KUKA KRL program: EPS_2_25252_SD6_A_20250910061732.src

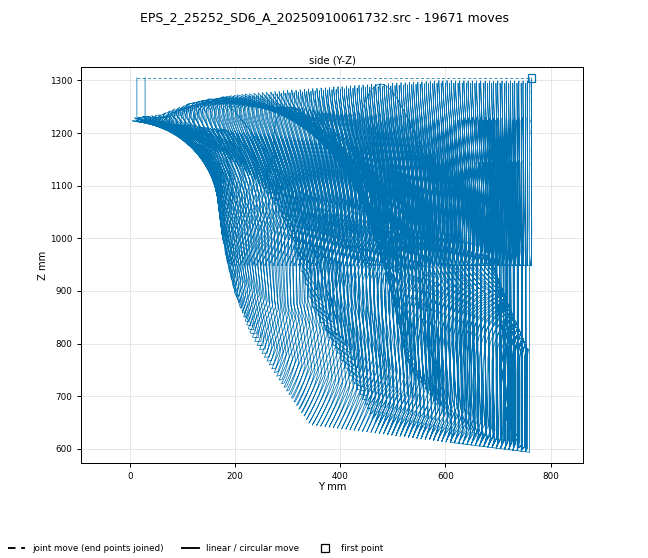
[picture p0: tool path of EPS_2_25252_SD6_A_20250910061732.src, 19671 of 19673 moves have a stored position in this frame; points joined in program order, loops and branches not executed]
&ACCESS RVP
&REL 4
&COMMENT QRS 19112012
&PARAM EDITMASK = *
DEF PART()
EXT BAS (BAS_COMMAND :IN,REAL :IN )
INT I
BAS (#INITMOV,0 )

;KUKA QRS Post kuka4.cps  Date:22-06-2017 !

File_ID=2834

QRS_PRE_INIT()

;Init var - Until changes are made in qrs_pre_init
Outlet_Square_prg=0
Inlet_1_Square_prg=0
Inlet_2_Square_prg=0
Inlet_3_Square_prg=0
Inlet_4_Square_prg=0
Inlet_5_Square_prg=0

Outlet_1={X 0.000, Y 582.000, Z 990.000, B 0.000, E1 0.000 }
Inlet_1={X 0.000, Y 651.840, Z 887.500, B 0.000, E1 181.000 }
Inlet_2={X 0.000, Y 582.000, Z 920.000, B 0.000, E1 273.000 }
Outlet_1_type=610
Inlet_1_type=299
Inlet_2_type=610
;QRS#1=Sidecore dimensions
;QRS#2=600-24" Concrete
;QRS#3=300-12" PVC SDR 35
;QRS#4=600-24" Concrete
;QRS#5=
;QRS#6=
;QRS#7=
;QRS#8=
;QRS#9=S306-34L
;QRS#10=16M PSX
;QRS#11=S306-34L
;QRS#12=
;QRS#13=
;QRS#14=
;QRS#15=
;QRS#16=1524x152x1753 5,75'
;QRS#17=EPS Height
;QRS#18=1295
;QRS#19=*
;QRS#20= UPDATED VERSION 22-06-2017
;QRS#21=*
Outlet_Square=0450
Inlet_1_Square=0150
Inlet_2_Square=0450
Inlet_3_Square=0
Inlet_4_Square=0
Inlet_5_Square=0
Mill_Square=1
Outlet_Square_Prg=264
Inlet_1_Square_prg=206
Inlet_2_Square_prg=264

QRS_INIT()

$ADVANCE=5

; T1
PTP {E1 176.595,E2 176.595}
PTP {X 0,Y 763.416,A -85,B 0,C 180,E1 176.595,E2 176.595,E3 0,E4 0,E5 0,E6 0}
QRS_SPEED_INIT()
LIN {X 0,Y 763.416,Z 1305,A -85,B 0,C 180,E1 176.595,E2 176.595,E3 0,E4 0,E5 0,E6 0} C_VEL
LIN {X 0,Y 763.416,Z 950.94,A -85,B 0,C 180,E1 176.595,E2 176.595} C_VEL
LIN {X 0,Y 763.526,Z 948.94,A -85,B 0,C 180,E1 176.744,E2 176.744} C_VEL
LIN {X 0,Y 763.879,Z 948.94,A -85,B 0,C 180,E1 177.187,E2 177.187} C_VEL
LIN {X 0,Y 763.856,Z 948.94,A -85,B 0,C 180,E1 184.692,E2 184.692} C_VEL
LIN {X 0,Y 763.844,Z 948.94,A -85,B 0,C 180,E1 192.28,E2 192.28} C_VEL
LIN {X 0,Y 763.822,Z 948.94,A -85,B 0,C 180,E1 200.096,E2 200.096} C_VEL
LIN {X 0,Y 763.802,Z 948.94,A -85,B 0,C 180,E1 208.326,E2 208.326} C_VEL
LIN {X 0,Y 762.908,Z 948.94,A -85,B 0,C 180,E1 213.344,E2 213.344} C_VEL
LIN {X 0,Y 763.801,Z 948.94,A -85,B 0,C 180,E1 214.936,E2 214.936} C_VEL
LIN {X 0,Y 762.569,Z 948.94,A -85,B 0,C 180,E1 217.327,E2 217.327} C_VEL
LIN {X 0,Y 763.787,Z 948.94,A -85,B 0,C 180,E1 222.132,E2 222.132} C_VEL
LIN {X 0,Y 763.6,Z 948.94,A -85,B 0,C 180,E1 222.571,E2 222.571} C_VEL
LIN {X 0,Y 763.857,Z 948.94,A -85,B 0,C 180,E1 230.259,E2 230.259} C_VEL
LIN {X 0,Y 763.749,Z 948.94,A -85,B 0,C 180,E1 236.564,E2 236.564} C_VEL
LIN {X 0,Y 763.497,Z 948.94,A -85,B 0,C 180,E1 237.308,E2 237.308} C_VEL
LIN {X 0,Y 763.827,Z 948.94,A -85,B 0,C 180,E1 243.397,E2 243.397} C_VEL
LIN {X 0,Y 763.404,Z 948.94,A -85,B 0,C 180,E1 243.594,E2 243.594} C_VEL
LIN {X 0,Y 763.701,Z 1010.798,A -85,B 0,C 180,E1 244.25,E2 244.25} C_VEL
LIN {X 0,Y 763.661,Z 1023.487,A -85,B 0,C 180,E1 244.413,E2 244.413} C_VEL
LIN {X 0,Y 763.555,Z 1034.565,A -85,B 0,C 180,E1 244.586,E2 244.586} C_VEL
LIN {X 0,Y 763.798,Z 1053.031,A -85,B 0,C 180,E1 244.967,E2 244.967} C_VEL
LIN {X 0,Y 763.799,Z 1068.002,A -85,B 0,C 180,E1 245.336,E2 245.336} C_VEL
LIN {X 0,Y 763.786,Z 1082.074,A -85,B 0,C 180,E1 245.738,E2 245.738} C_VEL
LIN {X 0,Y 763.598,Z 1095.558,A -85,B 0,C 180,E1 246.171,E2 246.171} C_VEL
LIN {X 0,Y 763.732,Z 1110.988,A -85,B 0,C 180,E1 246.751,E2 246.751} C_VEL
LIN {X 0,Y 763.705,Z 1123.304,A -85,B 0,C 180,E1 247.259,E2 247.259} C_VEL
LIN {X 0,Y 763.746,Z 1137.059,A -85,B 0,C 180,E1 247.894,E2 247.894} C_VEL
LIN {X 0,Y 763.694,Z 1150.472,A -85,B 0,C 180,E1 248.578,E2 248.578} C_VEL
LIN {X 0,Y 763.632,Z 1163.214,A -85,B 0,C 180,E1 249.293,E2 249.293} C_VEL
LIN {X 0,Y 763.454,Z 1174.901,A -85,B 0,C 180,E1 250.006,E2 250.006} C_VEL
LIN {X 0,Y 763.487,Z 1186.338,A -85,B 0,C 180,E1 250.774,E2 250.774} C_VEL
LIN {X 0,Y 763.678,Z 1195.926,A -85,B 0,C 180,E1 251.472,E2 251.472} C_VEL
LIN {X 0,Y 763.773,Z 1205.944,A -85,B 0,C 180,E1 252.258,E2 252.258} C_VEL
LIN {X 0,Y 763.425,Z 1217.367,A -85,B 0,C 180,E1 253.232,E2 253.232} C_VEL
LIN {X 0,Y 763.24,Z 1226.789,A -85,B 0,C 180,E1 254.111,E2 254.111} C_VEL
LIN {X 0,Y 763.374,Z 1235.4,A -85,B 0,C 180,E1 254.99,E2 254.99} C_VEL
LIN {X 0,Y 763.744,Z 1243.954,A -85,B 0,C 180,E1 255.948,E2 255.948} C_VEL
LIN {X 0,Y 763.788,Z 1247.786,A -85,B 0,C 180,E1 256.411,E2 256.411} C_VEL
LIN {X 0,Y 763.506,Z 1252.144,A -85,B 0,C 180,E1 256.944,E2 256.944} C_VEL
LIN {X 0,Y 763.029,Z 1259.656,A -85,B 0,C 180,E1 257.948,E2 257.948} C_VEL
LIN {X 0,Y 762.924,Z 1266.105,A -85,B 0,C 180,E1 258.904,E2 258.904} C_VEL
LIN {X 0,Y 763.387,Z 1273.197,A -85,B 0,C 180,E1 260.104,E2 260.104} C_VEL
LIN {X 0,Y 763.861,Z 1278.258,A -85,B 0,C 180,E1 261.06,E2 261.06} C_VEL
LIN {X 0,Y 763.274,Z 1282.688,A -85,B 0,C 180,E1 262.001,E2 262.001} C_VEL
LIN {X 0,Y 762.799,Z 1286.562,A -85,B 0,C 180,E1 262.943,E2 262.943} C_VEL
LIN {X 0,Y 762.692,Z 1288.341,A -85,B 0,C 180,E1 263.415,E2 263.415} C_VEL
LIN {X 0,Y 762.777,Z 1291.504,A -85,B 0,C 180,E1 264.36,E2 264.36} C_VEL
LIN {X 0,Y 763.282,Z 1294.069,A -85,B 0,C 180,E1 265.305,E2 265.305} C_VEL
LIN {X 0,Y 763.855,Z 1296.057,A -85,B 0,C 180,E1 266.211,E2 266.211} C_VEL
LIN {X 0,Y 763.535,Z 1297.167,A -85,B 0,C 180,E1 266.77,E2 266.77} C_VEL
LIN {X 0,Y 762.865,Z 1298.824,A -85,B 0,C 180,E1 267.936,E2 267.936} C_VEL
LIN {X 0,Y 762.698,Z 1299.723,A -85,B 0,C 180,E1 269.062,E2 269.062} C_VEL
LIN {X 0,Y 763.57,Z 1299.689,A -85,B 0,C 180,E1 270.939,E2 270.939} C_VEL
LIN {X 0,Y 763.743,Z 1299.172,A -85,B 0,C 180,E1 271.626,E2 271.626} C_VEL
LIN {X 0,Y 763.022,Z 1297.802,A -85,B 0,C 180,E1 272.817,E2 272.817} C_VEL
LIN {X 0,Y 762.7,Z 1296.172,A -85,B 0,C 180,E1 273.759,E2 273.759} C_VEL
LIN {X 0,Y 762.79,Z 1294.072,A -85,B 0,C 180,E1 274.7,E2 274.7} C_VEL
LIN {X 0,Y 763.256,Z 1291.49,A -85,B 0,C 180,E1 275.639,E2 275.639} C_VEL
LIN {X 0,Y 763.854,Z 1288.314,A -85,B 0,C 180,E1 276.577,E2 276.577} C_VEL
LIN {X 0,Y 763.331,Z 1284.657,A -85,B 0,C 180,E1 277.527,E2 277.527} C_VEL
LIN {X 0,Y 762.963,Z 1281.571,A -85,B 0,C 180,E1 278.241,E2 278.241} C_VEL
LIN {X 0,Y 762.777,Z 1278.249,A -85,B 0,C 180,E1 278.955,E2 278.955} C_VEL
LIN {X 0,Y 763.033,Z 1271.861,A -85,B 0,C 180,E1 280.142,E2 280.142} C_VEL
LIN {X 0,Y 763.586,Z 1266.091,A -85,B 0,C 180,E1 281.088,E2 281.088} C_VEL
LIN {X 0,Y 763.837,Z 1262.881,A -85,B 0,C 180,E1 281.563,E2 281.563} C_VEL
LIN {X 0,Y 763.471,Z 1257.055,A -85,B 0,C 180,E1 282.404,E2 282.404} C_VEL
LIN {X 0,Y 763.075,Z 1250.184,A -85,B 0,C 180,E1 283.313,E2 283.313} C_VEL
LIN {X 0,Y 763.016,Z 1242.631,A -85,B 0,C 180,E1 284.223,E2 284.223} C_VEL
LIN {X 0,Y 763.396,Z 1233.611,A -85,B 0,C 180,E1 285.201,E2 285.201} C_VEL
LIN {X 0,Y 763.805,Z 1223.978,A -85,B 0,C 180,E1 286.151,E2 286.151} C_VEL
LIN {X 0,Y 763.566,Z 1214.615,A -85,B 0,C 180,E1 287.012,E2 287.012} C_VEL
LIN {X 0,Y 763.309,Z 1204.368,A -85,B 0,C 180,E1 287.878,E2 287.878} C_VEL
LIN {X 0,Y 763.361,Z 1193.883,A -85,B 0,C 180,E1 288.687,E2 288.687} C_VEL
LIN {X 0,Y 763.618,Z 1182.933,A -85,B 0,C 180,E1 289.459,E2 289.459} C_VEL
LIN {X 0,Y 763.758,Z 1171.052,A -85,B 0,C 180,E1 290.229,E2 290.229} C_VEL
LIN {X 0,Y 763.669,Z 1158.921,A -85,B 0,C 180,E1 290.955,E2 290.955} C_VEL
LIN {X 0,Y 763.569,Z 1146.964,A -85,B 0,C 180,E1 291.612,E2 291.612} C_VEL
LIN {X 0,Y 763.634,Z 1134.379,A -85,B 0,C 180,E1 292.238,E2 292.238} C_VEL
LIN {X 0,Y 763.716,Z 1120.252,A -85,B 0,C 180,E1 292.87,E2 292.87} C_VEL
LIN {X 0,Y 763.734,Z 1110.933,A -85,B 0,C 180,E1 293.252,E2 293.252} C_VEL
LIN {X 0,Y 763.776,Z 1095.487,A -85,B 0,C 180,E1 293.826,E2 293.826} C_VEL
LIN {X 0,Y 763.739,Z 1080.093,A -85,B 0,C 180,E1 294.326,E2 294.326} C_VEL
LIN {X 0,Y 763.763,Z 1063.413,A -85,B 0,C 180,E1 294.785,E2 294.785} C_VEL
LIN {X 0,Y 763.546,Z 1049.599,A -85,B 0,C 180,E1 295.119,E2 295.119} C_VEL
LIN {X 0,Y 763.829,Z 1033.797,A -85,B 0,C 180,E1 295.417,E2 295.417} C_VEL
LIN {X 0,Y 763.825,Z 1018.657,A -85,B 0,C 180,E1 295.65,E2 295.65} C_VEL
LIN {X 0,Y 763.807,Z 1000.838,A -85,B 0,C 180,E1 295.857,E2 295.857} C_VEL
LIN {X 0,Y 763.398,Z 948.94,A -85,B 0,C 180,E1 296.405,E2 296.405} C_VEL
LIN {X 0,Y 763.703,Z 948.94,A -85,B 0,C 180,E1 296.465,E2 296.465} C_VEL
LIN {X 0,Y 763.627,Z 948.94,A -85,B 0,C 180,E1 297.495,E2 297.495} C_VEL
LIN {X 0,Y 763.6,Z 948.94,A -85,B 0,C 180,E1 298.335,E2 298.335} C_VEL
LIN {X 0,Y 763.684,Z 948.94,A -85,B 0,C 180,E1 299.853,E2 299.853} C_VEL
LIN {X 0,Y 763.798,Z 948.94,A -85,B 0,C 180,E1 307.257,E2 307.257} C_VEL
LIN {X 0,Y 762.303,Z 948.94,A -85,B 0,C 180,E1 312.462,E2 312.462} C_VEL
LIN {X 0,Y 763.54,Z 948.94,A -85,B 0,C 180,E1 314.733,E2 314.733} C_VEL
LIN {X 0,Y 763.758,Z 948.94,A -85,B 0,C 180,E1 315.284,E2 315.284} C_VEL
LIN {X 0,Y 763.727,Z 948.94,A -85,B 0,C 180,E1 323.303,E2 323.303} C_VEL
LIN {X 0,Y 762.819,Z 948.94,A -85,B 0,C 180,E1 325.013,E2 325.013} C_VEL
LIN {X 0,Y 763.876,Z 948.94,A -85,B 0,C 180,E1 330.979,E2 330.979} C_VEL
LIN {X 0,Y 762.688,Z 948.94,A -85,B 0,C 180,E1 331.215,E2 331.215} C_VEL
LIN {X 0,Y 762.37,Z 948.94,A -85,B 0,C 180,E1 331.237,E2 331.237} C_VEL
LIN {X 0,Y 762.335,Z 950.241,A -85,B 0,C 180,E1 331.271,E2 331.271} C_VEL
LIN {X 0,Y 763.361,Z 966.778,A -85,B 0,C 180,E1 331.573,E2 331.573} C_VEL
LIN {X 0,Y 763.732,Z 983.068,A -85,B 0,C 180,E1 331.92,E2 331.92} C_VEL
LIN {X 0,Y 763.791,Z 997.305,A -85,B 0,C 180,E1 332.271,E2 332.271} C_VEL
LIN {X 0,Y 763.798,Z 1012.281,A -85,B 0,C 180,E1 332.701,E2 332.701} C_VEL
LIN {X 0,Y 763.667,Z 1027.209,A -85,B 0,C 180,E1 333.189,E2 333.189} C_VEL
LIN {X 0,Y 763.708,Z 1041.233,A -85,B 0,C 180,E1 333.715,E2 333.715} C_VEL
LIN {X 0,Y 763.614,Z 1054.77,A -85,B 0,C 180,E1 334.278,E2 334.278} C_VEL
LIN {X 0,Y 763.605,Z 1067.742,A -85,B 0,C 180,E1 334.879,E2 334.879} C_VEL
LIN {X 0,Y 763.72,Z 1080.324,A -85,B 0,C 180,E1 335.525,E2 335.525} C_VEL
LIN {X 0,Y 763.702,Z 1092.995,A -85,B 0,C 180,E1 336.237,E2 336.237} C_VEL
LIN {X 0,Y 763.572,Z 1103.494,A -85,B 0,C 180,E1 336.871,E2 336.871} C_VEL
LIN {X 0,Y 763.366,Z 1114.975,A -85,B 0,C 180,E1 337.628,E2 337.628} C_VEL
LIN {X 0,Y 763.422,Z 1126.864,A -85,B 0,C 180,E1 338.494,E2 338.494} C_VEL
LIN {X 0,Y 763.687,Z 1137.376,A -85,B 0,C 180,E1 339.333,E2 339.333} C_VEL
LIN {X 0,Y 763.755,Z 1146.543,A -85,B 0,C 180,E1 340.119,E2 340.119} C_VEL
LIN {X 0,Y 763.366,Z 1156.466,A -85,B 0,C 180,E1 341.036,E2 341.036} C_VEL
LIN {X 0,Y 763.138,Z 1164.781,A -85,B 0,C 180,E1 341.872,E2 341.872} C_VEL
LIN {X 0,Y 763.296,Z 1173.673,A -85,B 0,C 180,E1 342.86,E2 342.86} C_VEL
LIN {X 0,Y 763.713,Z 1181.74,A -85,B 0,C 180,E1 343.848,E2 343.848} C_VEL
LIN {X 0,Y 763.782,Z 1185.725,A -85,B 0,C 180,E1 344.38,E2 344.38} C_VEL
LIN {X 0,Y 763.393,Z 1190.811,A -85,B 0,C 180,E1 345.08,E2 345.08} C_VEL
LIN {X 0,Y 763.022,Z 1195.576,A -85,B 0,C 180,E1 345.778,E2 345.778} C_VEL
LIN {X 0,Y 762.856,Z 1202.68,A -85,B 0,C 180,E1 346.955,E2 346.955} C_VEL
LIN {X 0,Y 763.206,Z 1207.972,A -85,B 0,C 180,E1 347.949,E2 347.949} C_VEL
LIN {X 0,Y 763.862,Z 1213.536,A -85,B 0,C 180,E1 349.155,E2 349.155} C_VEL
LIN {X 0,Y 763.274,Z 1217.354,A -85,B 0,C 180,E1 350.101,E2 350.101} C_VEL
LIN {X 0,Y 762.801,Z 1220.606,A -85,B 0,C 180,E1 351.046,E2 351.046} C_VEL
LIN {X 0,Y 762.674,Z 1222.073,A -85,B 0,C 180,E1 351.519,E2 351.519} C_VEL
LIN {X 0,Y 762.784,Z 1224.641,A -85,B 0,C 180,E1 352.469,E2 352.469} C_VEL
LIN {X 0,Y 763.298,Z 1226.62,A -85,B 0,C 180,E1 353.419,E2 353.419} C_VEL
LIN {X 0,Y 763.877,Z 1228.101,A -85,B 0,C 180,E1 354.367,E2 354.367} C_VEL
LIN {X 0,Y 763.297,Z 1229.174,A -85,B 0,C 180,E1 355.304,E2 355.304} C_VEL
LIN {X 0,Y 762.81,Z 1229.786,A -85,B 0,C 180,E1 356.243,E2 356.243} C_VEL
LIN {X 0,Y 762.699,Z 1229.932,A -85,B 0,C 180,E1 357.182,E2 357.182} C_VEL
LIN {X 0,Y 762.878,Z 1229.741,A -85,B 0,C 180,E1 357.815,E2 357.815} C_VEL
LIN {X 0,Y 763.571,Z 1228.757,A -85,B 0,C 180,E1 359.062,E2 359.062} C_VEL
LIN {X 0,Y 763.711,Z 1227.71,A -85,B 0,C 180,E1 359.812,E2 359.812} C_VEL
LIN {X 0,Y 763.226,Z 1226.472,A -85,B 0,C 180,E1 360.563,E2 360.563} C_VEL
LIN {X 0,Y 762.773,Z 1224.607,A -85,B 0,C 180,E1 361.456,E2 361.456} C_VEL
LIN {X 0,Y 762.819,Z 1220.763,A -85,B 0,C 180,E1 362.817,E2 362.817} C_VEL
LIN {X 0,Y 763.286,Z 1217.571,A -85,B 0,C 180,E1 363.755,E2 363.755} C_VEL
LIN {X 0,Y 763.871,Z 1213.785,A -85,B 0,C 180,E1 364.692,E2 364.692} C_VEL
LIN {X 0,Y 763.266,Z 1208.395,A -85,B 0,C 180,E1 365.873,E2 365.873} C_VEL
LIN {X 0,Y 762.935,Z 1202.109,A -85,B 0,C 180,E1 367.057,E2 367.057} C_VEL
LIN {X 0,Y 763.249,Z 1194.841,A -85,B 0,C 180,E1 368.237,E2 368.237} C_VEL
LIN {X 0,Y 763.726,Z 1188.367,A -85,B 0,C 180,E1 369.18,E2 369.18} C_VEL
LIN {X 0,Y 763.833,Z 1186.575,A -85,B 0,C 180,E1 369.416,E2 369.416} C_VEL
LIN {X 0,Y 763.53,Z 1181.216,A -85,B 0,C 180,E1 370.134,E2 370.134} C_VEL
LIN {X 0,Y 763.074,Z 1172.289,A -85,B 0,C 180,E1 371.214,E2 371.214} C_VEL
LIN {X 0,Y 763.072,Z 1163.507,A -85,B 0,C 180,E1 372.173,E2 372.173} C_VEL
LIN {X 0,Y 763.482,Z 1153.382,A -85,B 0,C 180,E1 373.167,E2 373.167} C_VEL
LIN {X 0,Y 763.794,Z 1145.374,A -85,B 0,C 180,E1 373.897,E2 373.897} C_VEL
LIN {X 0,Y 763.543,Z 1133.799,A -85,B 0,C 180,E1 374.872,E2 374.872} C_VEL
LIN {X 0,Y 763.312,Z 1124.099,A -85,B 0,C 180,E1 375.628,E2 375.628} C_VEL
LIN {X 0,Y 763.349,Z 1113.189,A -85,B 0,C 180,E1 376.404,E2 376.404} C_VEL
LIN {X 0,Y 763.612,Z 1100.958,A -85,B 0,C 180,E1 377.194,E2 377.194} C_VEL
LIN {X 0,Y 763.732,Z 1088.56,A -85,B 0,C 180,E1 377.929,E2 377.929} C_VEL
LIN {X 0,Y 763.702,Z 1076.06,A -85,B 0,C 180,E1 378.609,E2 378.609} C_VEL
LIN {X 0,Y 763.59,Z 1064.721,A -85,B 0,C 180,E1 379.179,E2 379.179} C_VEL
LIN {X 0,Y 763.625,Z 1050.751,A -85,B 0,C 180,E1 379.808,E2 379.808} C_VEL
LIN {X 0,Y 763.711,Z 1036.783,A -85,B 0,C 180,E1 380.369,E2 380.369} C_VEL
LIN {X 0,Y 763.667,Z 1025.67,A -85,B 0,C 180,E1 380.777,E2 380.777} C_VEL
LIN {X 0,Y 763.756,Z 1008.064,A -85,B 0,C 180,E1 381.338,E2 381.338} C_VEL
LIN {X 0,Y 763.736,Z 993.52,A -85,B 0,C 180,E1 381.739,E2 381.739} C_VEL
LIN {X 0,Y 763.708,Z 978.398,A -85,B 0,C 180,E1 382.093,E2 382.093} C_VEL
LIN {X 0,Y 763.357,Z 963.499,A -85,B 0,C 180,E1 382.393,E2 382.393} C_VEL
LIN {X 0,Y 762.407,Z 950.883,A -85,B 0,C 180,E1 382.628,E2 382.628} C_VEL
LIN {X 0,Y 762.139,Z 949.021,A -85,B 0,C 180,E1 382.661,E2 382.661} C_VEL
LIN {X 0,Y 763.124,Z 948.94,A -85,B 0,C 180,E1 382.74,E2 382.74} C_VEL
LIN {X 0,Y 763.665,Z 948.94,A -85,B 0,C 180,E1 383.269,E2 383.269} C_VEL
LIN {X 0,Y 763.828,Z 948.94,A -85,B 0,C 180,E1 388.325,E2 388.325} C_VEL
LIN {X 0,Y 762.698,Z 948.94,A -85,B 0,C 180,E1 394.994,E2 394.994} C_VEL
LIN {X 0,Y 763.702,Z 948.94,A -85,B 0,C 180,E1 396.695,E2 396.695} C_VEL
LIN {X 0,Y 763.721,Z 948.94,A -85,B 0,C 180,E1 404.719,E2 404.719} C_VEL
LIN {X 0,Y 763.507,Z 948.94,A -85,B 0,C 180,E1 405.265,E2 405.265} C_VEL
LIN {X 0,Y 762.431,Z 948.94,A -85,B 0,C 180,E1 410.388,E2 410.388} C_VEL
LIN {X 0,Y 763.801,Z 948.94,A -85,B 0,C 180,E1 412.743,E2 412.743} C_VEL
LIN {X 0,Y 763.669,Z 948.94,A -85,B 0,C 180,E1 420.149,E2 420.149} C_VEL
LIN {X 0,Y 762.955,Z 948.94,A -85,B 0,C 180,E1 421.639,E2 421.639} C_VEL
LIN {X 0,Y 763.83,Z 948.94,A -85,B 0,C 180,E1 427.894,E2 427.894} C_VEL
LIN {X 0,Y 763.858,Z 948.94,A -85,B 0,C 180,E1 434.777,E2 434.777} C_VEL
LIN {X 0,Y 763.313,Z 948.94,A -85,B 0,C 180,E1 434.94,E2 434.94} C_VEL
LIN {X 0,Y 762.376,Z 948.94,A -85,B 0,C 180,E1 435.024,E2 435.024} C_VEL
LIN {X 0,Y 763.453,Z 975.866,A -85,B 0,C 180,E1 435.303,E2 435.303} C_VEL
LIN {X 0,Y 763.818,Z 998.319,A -85,B 0,C 180,E1 435.532,E2 435.532} C_VEL
LIN {X 0,Y 763.817,Z 1010.228,A -85,B 0,C 180,E1 435.708,E2 435.708} C_VEL
LIN {X 0,Y 763.804,Z 1018.714,A -85,B 0,C 180,E1 435.874,E2 435.874} C_VEL
LIN {X 0,Y 763.805,Z 1028.192,A -85,B 0,C 180,E1 436.1,E2 436.1} C_VEL
LIN {X 0,Y 763.731,Z 1036.369,A -85,B 0,C 180,E1 436.329,E2 436.329} C_VEL
LIN {X 0,Y 763.74,Z 1044.631,A -85,B 0,C 180,E1 436.598,E2 436.598} C_VEL
LIN {X 0,Y 763.845,Z 1054.622,A -85,B 0,C 180,E1 436.974,E2 436.974} C_VEL
LIN {X 0,Y 763.835,Z 1063.932,A -85,B 0,C 180,E1 437.383,E2 437.383} C_VEL
LIN {X 0,Y 763.698,Z 1071.923,A -85,B 0,C 180,E1 437.777,E2 437.777} C_VEL
LIN {X 0,Y 763.546,Z 1079.501,A -85,B 0,C 180,E1 438.194,E2 438.194} C_VEL
LIN {X 0,Y 763.575,Z 1087.281,A -85,B 0,C 180,E1 438.673,E2 438.673} C_VEL
LIN {X 0,Y 763.799,Z 1095.832,A -85,B 0,C 180,E1 439.273,E2 439.273} C_VEL
LIN {X 0,Y 763.835,Z 1101.944,A -85,B 0,C 180,E1 439.75,E2 439.75} C_VEL
LIN {X 0,Y 763.6,Z 1107.496,A -85,B 0,C 180,E1 440.223,E2 440.223} C_VEL
LIN {X 0,Y 763.321,Z 1112.557,A -85,B 0,C 180,E1 440.695,E2 440.695} C_VEL
LIN {X 0,Y 763.183,Z 1117.18,A -85,B 0,C 180,E1 441.168,E2 441.168} C_VEL
LIN {X 0,Y 763.261,Z 1121.403,A -85,B 0,C 180,E1 441.644,E2 441.644} C_VEL
LIN {X 0,Y 763.56,Z 1126.164,A -85,B 0,C 180,E1 442.239,E2 442.239} C_VEL
LIN {X 0,Y 763.801,Z 1129.593,A -85,B 0,C 180,E1 442.714,E2 442.714} C_VEL
LIN {X 0,Y 763.871,Z 1131.208,A -85,B 0,C 180,E1 442.951,E2 442.951} C_VEL
LIN {X 0,Y 763.472,Z 1135.557,A -85,B 0,C 180,E1 443.655,E2 443.655} C_VEL
LIN {X 0,Y 763.096,Z 1139.231,A -85,B 0,C 180,E1 444.36,E2 444.36} C_VEL
LIN {X 0,Y 763.009,Z 1141.39,A -85,B 0,C 180,E1 444.831,E2 444.831} C_VEL
LIN {X 0,Y 763.112,Z 1143.271,A -85,B 0,C 180,E1 445.302,E2 445.302} C_VEL
LIN {X 0,Y 763.388,Z 1145.04,A -85,B 0,C 180,E1 445.823,E2 445.823} C_VEL
LIN {X 0,Y 763.774,Z 1146.85,A -85,B 0,C 180,E1 446.466,E2 446.466} C_VEL
LIN {X 0,Y 763.607,Z 1148.403,A -85,B 0,C 180,E1 447.185,E2 447.185} C_VEL
LIN {X 0,Y 763.131,Z 1149.434,A -85,B 0,C 180,E1 447.934,E2 447.934} C_VEL
LIN {X 0,Y 762.969,Z 1149.77,A -85,B 0,C 180,E1 448.309,E2 448.309} C_VEL
LIN {X 0,Y 762.962,Z 1149.961,A -85,B 0,C 180,E1 449.06,E2 449.06} C_VEL
LIN {X 0,Y 763.329,Z 1149.57,A -85,B 0,C 180,E1 449.811,E2 449.811} C_VEL
LIN {X 0,Y 763.801,Z 1148.636,A -85,B 0,C 180,E1 450.561,E2 450.561} C_VEL
LIN {X 0,Y 763.769,Z 1147.968,A -85,B 0,C 180,E1 450.936,E2 450.936} C_VEL
LIN {X 0,Y 763.177,Z 1145.441,A -85,B 0,C 180,E1 451.97,E2 451.97} C_VEL
LIN {X 0,Y 763.031,Z 1143.772,A -85,B 0,C 180,E1 452.471,E2 452.471} C_VEL
LIN {X 0,Y 763.126,Z 1141.244,A -85,B 0,C 180,E1 453.114,E2 453.114} C_VEL
LIN {X 0,Y 763.441,Z 1138.352,A -85,B 0,C 180,E1 453.733,E2 453.733} C_VEL
LIN {X 0,Y 763.825,Z 1134.861,A -85,B 0,C 180,E1 454.371,E2 454.371} C_VEL
LIN {X 0,Y 763.669,Z 1131.439,A -85,B 0,C 180,E1 454.927,E2 454.927} C_VEL
LIN {X 0,Y 763.323,Z 1126.447,A -85,B 0,C 180,E1 455.636,E2 455.636} C_VEL
LIN {X 0,Y 763.231,Z 1120.749,A -85,B 0,C 180,E1 456.344,E2 456.344} C_VEL
LIN {X 0,Y 763.532,Z 1114.219,A -85,B 0,C 180,E1 457.05,E2 457.05} C_VEL
LIN {X 0,Y 763.832,Z 1108.014,A -85,B 0,C 180,E1 457.638,E2 457.638} C_VEL
LIN {X 0,Y 763.786,Z 1102.54,A -85,B 0,C 180,E1 458.112,E2 458.112} C_VEL
LIN {X 0,Y 763.575,Z 1096.526,A -85,B 0,C 180,E1 458.588,E2 458.588} C_VEL
LIN {X 0,Y 763.441,Z 1089.89,A -85,B 0,C 180,E1 459.064,E2 459.064} C_VEL
LIN {X 0,Y 763.556,Z 1081.564,A -85,B 0,C 180,E1 459.597,E2 459.597} C_VEL
LIN {X 0,Y 763.796,Z 1073.109,A -85,B 0,C 180,E1 460.07,E2 460.07} C_VEL
LIN {X 0,Y 763.853,Z 1066.053,A -85,B 0,C 180,E1 460.426,E2 460.426} C_VEL
LIN {X 0,Y 763.8,Z 1058.187,A -85,B 0,C 180,E1 460.784,E2 460.784} C_VEL
LIN {X 0,Y 763.629,Z 1049.304,A -85,B 0,C 180,E1 461.145,E2 461.145} C_VEL
LIN {X 0,Y 763.644,Z 1038.984,A -85,B 0,C 180,E1 461.503,E2 461.503} C_VEL
LIN {X 0,Y 763.804,Z 1029.717,A -85,B 0,C 180,E1 461.77,E2 461.77} C_VEL
LIN {X 0,Y 763.777,Z 1020.573,A -85,B 0,C 180,E1 461.995,E2 461.995} C_VEL
LIN {X 0,Y 763.848,Z 1011.303,A -85,B 0,C 180,E1 462.181,E2 462.181} C_VEL
LIN {X 0,Y 763.833,Z 1000.704,A -85,B 0,C 180,E1 462.349,E2 462.349} C_VEL
LIN {X 0,Y 763.809,Z 984.227,A -85,B 0,C 180,E1 462.521,E2 462.521} C_VEL
LIN {X 0,Y 763.331,Z 953.121,A -85,B 0,C 180,E1 462.825,E2 462.825} C_VEL
LIN {X 0,Y 763.254,Z 948.94,A -85,B 0,C 180,E1 462.872,E2 462.872} C_VEL
LIN {X 0,Y 763.703,Z 948.94,A -85,B 0,C 180,E1 462.95,E2 462.95} C_VEL
LIN {X 0,Y 763.603,Z 948.94,A -85,B 0,C 180,E1 463.37,E2 463.37} C_VEL
LIN {X 0,Y 763.824,Z 948.94,A -85,B 0,C 180,E1 470.094,E2 470.094} C_VEL
LIN {X 0,Y 763.807,Z 948.94,A -85,B 0,C 180,E1 478.324,E2 478.324} C_VEL
LIN {X 0,Y 761.983,Z 948.94,A -85,B 0,C 180,E1 482.765,E2 482.765} C_VEL
LIN {X 0,Y 762.706,Z 948.94,A -85,B 0,C 180,E1 484.991,E2 484.991} C_VEL
LIN {X 0,Y 763.719,Z 948.94,A -85,B 0,C 180,E1 486.697,E2 486.697} C_VEL
LIN {X 0,Y 763.746,Z 948.94,A -85,B 0,C 180,E1 494.714,E2 494.714} C_VEL
LIN {X 0,Y 763.531,Z 948.94,A -85,B 0,C 180,E1 495.267,E2 495.267} C_VEL
LIN {X 0,Y 762.429,Z 948.94,A -85,B 0,C 180,E1 500.385,E2 500.385} C_VEL
LIN {X 0,Y 763.793,Z 948.94,A -85,B 0,C 180,E1 502.743,E2 502.743} C_VEL
LIN {X 0,Y 763.668,Z 948.94,A -85,B 0,C 180,E1 510.145,E2 510.145} C_VEL
LIN {X 0,Y 762.96,Z 948.94,A -85,B 0,C 180,E1 511.64,E2 511.64} C_VEL
LIN {X 0,Y 763.826,Z 948.94,A -85,B 0,C 180,E1 517.895,E2 517.895} C_VEL
LIN {X 0,Y 763.489,Z 948.94,A -85,B 0,C 180,E1 524.95,E2 524.95} C_VEL
LIN {X 0,Y 763.685,Z 948.94,A -85,B 0,C 180,E1 525.791,E2 525.791} C_VEL
LIN {X 0,Y 763.849,Z 948.94,A -85,B 0,C 180,E1 529.632,E2 529.632} C_VEL
LIN {X 0,Y 763.526,Z 948.94,A -85,B 0,C 180,E1 536.744,E2 536.744} C_VEL
LIN {X 0,Y 754.559,Z 948.94,A -85,B 0,C 180,E1 539.344,E2 539.344} C_VEL
LIN {X 0,Y 754.729,Z 948.94,A -85,B 0,C 180,E1 546.339,E2 546.339} C_VEL
LIN {X 0,Y 754.988,Z 948.94,A -85,B 0,C 180,E1 553.356,E2 553.356} C_VEL
LIN {X 0,Y 755.078,Z 948.94,A -85,B 0,C 180,E1 560.952,E2 560.952} C_VEL
LIN {X 0,Y 755.072,Z 948.94,A -85,B 0,C 180,E1 569.491,E2 569.491} C_VEL
LIN {X 0,Y 754.903,Z 948.94,A -85,B 0,C 180,E1 576.365,E2 576.365} C_VEL
LIN {X 0,Y 755.336,Z 948.94,A -85,B 0,C 180,E1 582.888,E2 582.888} C_VEL
LIN {X 0,Y 755.509,Z 948.94,A -85,B 0,C 180,E1 590.794,E2 590.794} C_VEL
LIN {X 0,Y 755.189,Z 948.94,A -85,B 0,C 180,E1 597.865,E2 597.865} C_VEL
LIN {X 0,Y 755.986,Z 950.766,A -85,B 0,C 180,E1 603.335,E2 603.335} C_VEL
LIN {X 0,Y 756.522,Z 1050.329,A -85,B 0,C 180,E1 604.647,E2 604.647} C_VEL
LIN {X 0,Y 756.258,Z 1115.341,A -85,B 0,C 180,E1 606.688,E2 606.688} C_VEL
LIN {X 0,Y 755.771,Z 1175.676,A -85,B 0,C 180,E1 609.845,E2 609.845} C_VEL
LIN {X 0,Y 755.412,Z 1225.871,A -85,B 0,C 180,E1 613.848,E2 613.848} C_VEL
LIN {X 0,Y 755.043,Z 1261.823,A -85,B 0,C 180,E1 618.142,E2 618.142} C_VEL
LIN {X 0,Y 755.002,Z 1285.187,A -85,B 0,C 180,E1 622.523,E2 622.523} C_VEL
LIN {X 0,Y 755.286,Z 1297.813,A -85,B 0,C 180,E1 627.15,E2 627.15} C_VEL
LIN {X 0,Y 755.662,Z 1299.126,A -85,B 0,C 180,E1 631.754,E2 631.754} C_VEL
LIN {X 0,Y 755.652,Z 1287.259,A -85,B 0,C 180,E1 636.948,E2 636.948} C_VEL
LIN {X 0,Y 755.604,Z 1259.469,A -85,B 0,C 180,E1 642.201,E2 642.201} C_VEL
LIN {X 0,Y 755.774,Z 1218.868,A -85,B 0,C 180,E1 646.803,E2 646.803} C_VEL
LIN {X 0,Y 756.05,Z 1166.963,A -85,B 0,C 180,E1 650.695,E2 650.695} C_VEL
LIN {X 0,Y 756.349,Z 1106.488,A -85,B 0,C 180,E1 653.668,E2 653.668} C_VEL
LIN {X 0,Y 756.515,Z 1039.409,A -85,B 0,C 180,E1 655.575,E2 655.575} C_VEL
LIN {X 0,Y 755.673,Z 948.94,A -85,B 0,C 180,E1 656.755,E2 656.755} C_VEL
LIN {X 0,Y 754.178,Z 948.94,A -85,B 0,C 180,E1 663.624,E2 663.624} C_VEL
LIN {X 0,Y 754.493,Z 948.94,A -85,B 0,C 180,E1 669.258,E2 669.258} C_VEL
LIN {X 0,Y 755.064,Z 948.94,A -85,B 0,C 180,E1 676.107,E2 676.107} C_VEL
LIN {X 0,Y 755.02,Z 948.94,A -85,B 0,C 180,E1 684.525,E2 684.525} C_VEL
LIN {X 0,Y 755.078,Z 949.483,A -85,B 0,C 180,E1 690.997,E2 690.997} C_VEL
LIN {X 0,Y 756.378,Z 1018.428,A -85,B 0,C 180,E1 692.648,E2 692.648} C_VEL
LIN {X 0,Y 756.117,Z 1080.659,A -85,B 0,C 180,E1 695.318,E2 695.318} C_VEL
LIN {X 0,Y 755.833,Z 1136.369,A -85,B 0,C 180,E1 699.058,E2 699.058} C_VEL
LIN {X 0,Y 755.639,Z 1180.363,A -85,B 0,C 180,E1 703.529,E2 703.529} C_VEL
LIN {X 0,Y 755.444,Z 1210.603,A -85,B 0,C 180,E1 708.421,E2 708.421} C_VEL
LIN {X 0,Y 755.447,Z 1227.166,A -85,B 0,C 180,E1 713.667,E2 713.667} C_VEL
LIN {X 0,Y 755.103,Z 1229.503,A -85,B 0,C 180,E1 718.283,E2 718.283} C_VEL
LIN {X 0,Y 755.128,Z 1218.8,A -85,B 0,C 180,E1 723.468,E2 723.468} C_VEL
LIN {X 0,Y 755.357,Z 1194.629,A -85,B 0,C 180,E1 728.388,E2 728.388} C_VEL
LIN {X 0,Y 755.603,Z 1155.266,A -85,B 0,C 180,E1 733.164,E2 733.164} C_VEL
LIN {X 0,Y 755.884,Z 1104.369,A -85,B 0,C 180,E1 737.193,E2 737.193} C_VEL
LIN {X 0,Y 756.207,Z 1043.498,A -85,B 0,C 180,E1 740.346,E2 740.346} C_VEL
LIN {X 0,Y 756.427,Z 978.742,A -85,B 0,C 180,E1 742.345,E2 742.345} C_VEL
LIN {X 0,Y 755.452,Z 948.94,A -85,B 0,C 180,E1 743.078,E2 743.078} C_VEL
LIN {X 0,Y 754.85,Z 948.94,A -85,B 0,C 180,E1 749.527,E2 749.527} C_VEL
LIN {X 0,Y 754.795,Z 948.94,A -85,B 0,C 180,E1 757.844,E2 757.844} C_VEL
LIN {X 0,Y 754.95,Z 948.94,A -85,B 0,C 180,E1 766.063,E2 766.063} C_VEL
LIN {X 0,Y 755.132,Z 948.94,A -85,B 0,C 180,E1 773.613,E2 773.613} C_VEL
LIN {X 0,Y 754.882,Z 948.94,A -85,B 0,C 180,E1 781.782,E2 781.782} C_VEL
LIN {X 0,Y 754.922,Z 948.94,A -85,B 0,C 180,E1 789.377,E2 789.377} C_VEL
LIN {X 0,Y 754.639,Z 950.118,A -85,B 0,C 180,E1 794.893,E2 794.893} C_VEL
LIN {X 0,Y 756.032,Z 1025.236,A -85,B 0,C 180,E1 795.887,E2 795.887} C_VEL
LIN {X 0,Y 755.828,Z 1071.872,A -85,B 0,C 180,E1 797.656,E2 797.656} C_VEL
LIN {X 0,Y 755.483,Z 1110.797,A -85,B 0,C 180,E1 800.434,E2 800.434} C_VEL
LIN {X 0,Y 755.339,Z 1137.046,A -85,B 0,C 180,E1 803.878,E2 803.878} C_VEL
LIN {X 0,Y 755.646,Z 1148.306,A -85,B 0,C 180,E1 807.094,E2 807.094} C_VEL
LIN {X 0,Y 755.664,Z 1147.673,A -85,B 0,C 180,E1 811.122,E2 811.122} C_VEL
LIN {X 0,Y 755.709,Z 1132.236,A -85,B 0,C 180,E1 814.866,E2 814.866} C_VEL
LIN {X 0,Y 755.816,Z 1102.715,A -85,B 0,C 180,E1 818.195,E2 818.195} C_VEL
LIN {X 0,Y 755.985,Z 1061.969,A -85,B 0,C 180,E1 820.743,E2 820.743} C_VEL
LIN {X 0,Y 756.05,Z 1014.246,A -85,B 0,C 180,E1 822.265,E2 822.265} C_VEL
LIN {X 0,Y 755.681,Z 948.94,A -85,B 0,C 180,E1 823.082,E2 823.082} C_VEL
LIN {X 0,Y 755.185,Z 948.94,A -85,B 0,C 180,E1 830.808,E2 830.808} C_VEL
LIN {X 0,Y 754.898,Z 948.94,A -85,B 0,C 180,E1 839.467,E2 839.467} C_VEL
LIN {X 0,Y 754.847,Z 948.94,A -85,B 0,C 180,E1 847.775,E2 847.775} C_VEL
LIN {X 0,Y 754.955,Z 948.94,A -85,B 0,C 180,E1 856.068,E2 856.068} C_VEL
LIN {X 0,Y 755.119,Z 948.94,A -85,B 0,C 180,E1 863.619,E2 863.619} C_VEL
LIN {X 0,Y 754.889,Z 948.94,A -85,B 0,C 180,E1 871.791,E2 871.791} C_VEL
LIN {X 0,Y 754.785,Z 948.94,A -85,B 0,C 180,E1 879.384,E2 879.384} C_VEL
LIN {X 0,Y 755.395,Z 948.94,A -85,B 0,C 180,E1 886.821,E2 886.821} C_VEL
LIN {X 0,Y 754.227,Z 948.94,A -85,B 0,C 180,E1 893.634,E2 893.634} C_VEL
LIN {X 0,Y 755.089,Z 948.94,A -85,B 0,C 180,E1 898.261,E2 898.261} C_VEL
LIN {X 0,Y 754.559,Z 948.94,A -85,B 0,C 180,E1 899.344,E2 899.344} C_VEL
LIN {X 0,Y 746.381,Z 948.94,A -85,B 0,C 180,E1 901.974,E2 901.974} C_VEL
LIN {X 0,Y 746.272,Z 948.94,A -85,B 0,C 180,E1 907.585,E2 907.585} C_VEL
LIN {X 0,Y 746.888,Z 948.94,A -85,B 0,C 180,E1 913.503,E2 913.503} C_VEL
LIN {X 0,Y 747.18,Z 948.94,A -85,B 0,C 180,E1 920.811,E2 920.811} C_VEL
LIN {X 0,Y 747.51,Z 948.94,A -85,B 0,C 180,E1 928.487,E2 928.487} C_VEL
LIN {X 0,Y 747.468,Z 948.94,A -85,B 0,C 180,E1 935.347,E2 935.347} C_VEL
LIN {X 0,Y 747.347,Z 948.94,A -85,B 0,C 180,E1 942.856,E2 942.856} C_VEL
LIN {X 0,Y 747.013,Z 948.94,A -85,B 0,C 180,E1 951.758,E2 951.758} C_VEL
LIN {X 0,Y 746.804,Z 948.94,A -85,B 0,C 180,E1 958.83,E2 958.83} C_VEL
LIN {X 0,Y 747.641,Z 949.984,A -85,B 0,C 180,E1 963.005,E2 963.005} C_VEL
LIN {X 0,Y 749.261,Z 1051.983,A -85,B 0,C 180,E1 964.421,E2 964.421} C_VEL
LIN {X 0,Y 748.787,Z 1117.47,A -85,B 0,C 180,E1 966.53,E2 966.53} C_VEL
LIN {X 0,Y 748.074,Z 1176.827,A -85,B 0,C 180,E1 969.706,E2 969.706} C_VEL
LIN {X 0,Y 747.578,Z 1225.875,A -85,B 0,C 180,E1 973.674,E2 973.674} C_VEL
LIN {X 0,Y 747.109,Z 1261.826,A -85,B 0,C 180,E1 978.015,E2 978.015} C_VEL
LIN {X 0,Y 747.042,Z 1285.188,A -85,B 0,C 180,E1 982.443,E2 982.443} C_VEL
LIN {X 0,Y 747.327,Z 1297.816,A -85,B 0,C 180,E1 987.119,E2 987.119} C_VEL
LIN {X 0,Y 747.638,Z 1299.129,A -85,B 0,C 180,E1 991.773,E2 991.773} C_VEL
LIN {X 0,Y 747.608,Z 1287.258,A -85,B 0,C 180,E1 997.023,E2 997.023} C_VEL
LIN {X 0,Y 747.63,Z 1259.472,A -85,B 0,C 180,E1 1002.333,E2 1002.333} C_VEL
LIN {X 0,Y 747.931,Z 1218.873,A -85,B 0,C 180,E1 1006.985,E2 1006.985} C_VEL
LIN {X 0,Y 748.38,Z 1167.417,A -85,B 0,C 180,E1 1010.89,E2 1010.89} C_VEL
LIN {X 0,Y 748.918,Z 1106.901,A -85,B 0,C 180,E1 1013.901,E2 1013.901} C_VEL
LIN {X 0,Y 749.283,Z 1040.606,A -85,B 0,C 180,E1 1015.816,E2 1015.816} C_VEL
LIN {X 0,Y 747.638,Z 948.94,A -85,B 0,C 180,E1 1017.046,E2 1017.046} C_VEL
LIN {X 0,Y 746.6,Z 948.94,A -85,B 0,C 180,E1 1025.429,E2 1025.429} C_VEL
LIN {X 0,Y 746.476,Z 948.94,A -85,B 0,C 180,E1 1032.954,E2 1032.954} C_VEL
LIN {X 0,Y 746.091,Z 948.94,A -85,B 0,C 180,E1 1037.968,E2 1037.968} C_VEL
LIN {X 0,Y 747.003,Z 948.94,A -85,B 0,C 180,E1 1044.628,E2 1044.628} C_VEL
LIN {X 0,Y 747.821,Z 950.432,A -85,B 0,C 180,E1 1050.738,E2 1050.738} C_VEL
LIN {X 0,Y 749,Z 1020.318,A -85,B 0,C 180,E1 1052.455,E2 1052.455} C_VEL
LIN {X 0,Y 748.509,Z 1081.829,A -85,B 0,C 180,E1 1055.153,E2 1055.153} C_VEL
LIN {X 0,Y 748.016,Z 1137.068,A -85,B 0,C 180,E1 1058.925,E2 1058.925} C_VEL
LIN {X 0,Y 747.722,Z 1181.279,A -85,B 0,C 180,E1 1063.502,E2 1063.502} C_VEL
LIN {X 0,Y 747.558,Z 1211.812,A -85,B 0,C 180,E1 1068.594,E2 1068.594} C_VEL
LIN {X 0,Y 747.393,Z 1227.12,A -85,B 0,C 180,E1 1073.598,E2 1073.598} C_VEL
LIN {X 0,Y 747.112,Z 1229.534,A -85,B 0,C 180,E1 1078.265,E2 1078.265} C_VEL
LIN {X 0,Y 747.175,Z 1218.908,A -85,B 0,C 180,E1 1083.505,E2 1083.505} C_VEL
LIN {X 0,Y 747.446,Z 1194.849,A -85,B 0,C 180,E1 1088.478,E2 1088.478} C_VEL
LIN {X 0,Y 747.759,Z 1155.602,A -85,B 0,C 180,E1 1093.304,E2 1093.304} C_VEL
LIN {X 0,Y 748.238,Z 1104.411,A -85,B 0,C 180,E1 1097.406,E2 1097.406} C_VEL
LIN {X 0,Y 748.748,Z 1044.343,A -85,B 0,C 180,E1 1100.557,E2 1100.557} C_VEL
LIN {X 0,Y 749.144,Z 978.027,A -85,B 0,C 180,E1 1102.625,E2 1102.625} C_VEL
LIN {X 0,Y 747.413,Z 948.94,A -85,B 0,C 180,E1 1103.34,E2 1103.34} C_VEL
LIN {X 0,Y 746.624,Z 948.94,A -85,B 0,C 180,E1 1109.885,E2 1109.885} C_VEL
LIN {X 0,Y 747.269,Z 948.94,A -85,B 0,C 180,E1 1116.826,E2 1116.826} C_VEL
LIN {X 0,Y 747.307,Z 948.94,A -85,B 0,C 180,E1 1125.496,E2 1125.496} C_VEL
LIN {X 0,Y 747.216,Z 948.94,A -85,B 0,C 180,E1 1133.375,E2 1133.375} C_VEL
LIN {X 0,Y 747.003,Z 948.94,A -85,B 0,C 180,E1 1141.457,E2 1141.457} C_VEL
LIN {X 0,Y 747.016,Z 948.94,A -85,B 0,C 180,E1 1149.149,E2 1149.149} C_VEL
LIN {X 0,Y 746.892,Z 950.692,A -85,B 0,C 180,E1 1154.75,E2 1154.75} C_VEL
LIN {X 0,Y 748.223,Z 1024.79,A -85,B 0,C 180,E1 1155.737,E2 1155.737} C_VEL
LIN {X 0,Y 748.004,Z 1070.773,A -85,B 0,C 180,E1 1157.477,E2 1157.477} C_VEL
LIN {X 0,Y 747.676,Z 1109.141,A -85,B 0,C 180,E1 1160.186,E2 1160.186} C_VEL
LIN {X 0,Y 747.527,Z 1135.667,A -85,B 0,C 180,E1 1163.562,E2 1163.562} C_VEL
LIN {X 0,Y 747.68,Z 1148.283,A -85,B 0,C 180,E1 1167.063,E2 1167.063} C_VEL
LIN {X 0,Y 747.654,Z 1147.696,A -85,B 0,C 180,E1 1171.134,E2 1171.134} C_VEL
LIN {X 0,Y 747.695,Z 1132.305,A -85,B 0,C 180,E1 1174.919,E2 1174.919} C_VEL
LIN {X 0,Y 747.864,Z 1102.854,A -85,B 0,C 180,E1 1178.282,E2 1178.282} C_VEL
LIN {X 0,Y 748.116,Z 1061.958,A -85,B 0,C 180,E1 1180.869,E2 1180.869} C_VEL
LIN {X 0,Y 748.269,Z 1015.292,A -85,B 0,C 180,E1 1182.386,E2 1182.386} C_VEL
LIN {X 0,Y 747.64,Z 948.94,A -85,B 0,C 180,E1 1183.289,E2 1183.289} C_VEL
LIN {X 0,Y 747.221,Z 948.94,A -85,B 0,C 180,E1 1190.784,E2 1190.784} C_VEL
LIN {X 0,Y 747.445,Z 948.94,A -85,B 0,C 180,E1 1198.459,E2 1198.459} C_VEL
LIN {X 0,Y 747.266,Z 948.94,A -85,B 0,C 180,E1 1206.761,E2 1206.761} C_VEL
LIN {X 0,Y 746.925,Z 948.94,A -85,B 0,C 180,E1 1216.106,E2 1216.106} C_VEL
LIN {X 0,Y 747.207,Z 948.94,A -85,B 0,C 180,E1 1223.281,E2 1223.281} C_VEL
LIN {X 0,Y 746.774,Z 948.94,A -85,B 0,C 180,E1 1232.045,E2 1232.045} C_VEL
LIN {X 0,Y 746.949,Z 948.94,A -85,B 0,C 180,E1 1239.158,E2 1239.158} C_VEL
LIN {X 0,Y 747.37,Z 948.94,A -85,B 0,C 180,E1 1247.676,E2 1247.676} C_VEL
LIN {X 0,Y 747.78,Z 948.94,A -85,B 0,C 180,E1 1257.08,E2 1257.08} C_VEL
LIN {X 0,Y 746.381,Z 948.94,A -85,B 0,C 180,E1 1261.974,E2 1261.974} C_VEL
LIN {X 0,Y 739.31,Z 948.94,A -85,B 0,C 180,E1 1264.655,E2 1264.655} C_VEL
LIN {X 0,Y 738.82,Z 948.94,A -85,B 0,C 180,E1 1273.654,E2 1273.654} C_VEL
LIN {X 0,Y 739.007,Z 948.94,A -85,B 0,C 180,E1 1281.052,E2 1281.052} C_VEL
LIN {X 0,Y 739.105,Z 948.94,A -85,B 0,C 180,E1 1289.314,E2 1289.314} C_VEL
LIN {X 0,Y 739.146,Z 948.94,A -85,B 0,C 180,E1 1295.873,E2 1295.873} C_VEL
LIN {X 0,Y 738.923,Z 948.94,A -85,B 0,C 180,E1 1303.465,E2 1303.465} C_VEL
LIN {X 0,Y 739.186,Z 948.94,A -85,B 0,C 180,E1 1311.278,E2 1311.278} C_VEL
LIN {X 0,Y 738.902,Z 948.94,A -85,B 0,C 180,E1 1318.459,E2 1318.459} C_VEL
LIN {X 0,Y 739.463,Z 950.322,A -85,B 0,C 180,E1 1322.686,E2 1322.686} C_VEL
LIN {X 0,Y 742.066,Z 973.283,A -85,B 0,C 180,E1 1323.034,E2 1323.034} C_VEL
LIN {X 0,Y 741.99,Z 1053.627,A -85,B 0,C 180,E1 1324.192,E2 1324.192} C_VEL
LIN {X 0,Y 741.327,Z 1118.969,A -85,B 0,C 180,E1 1326.343,E2 1326.343} C_VEL
LIN {X 0,Y 740.375,Z 1177.978,A -85,B 0,C 180,E1 1329.564,E2 1329.564} C_VEL
LIN {X 0,Y 739.686,Z 1227.353,A -85,B 0,C 180,E1 1333.648,E2 1333.648} C_VEL
LIN {X 0,Y 739.128,Z 1263.796,A -85,B 0,C 180,E1 1338.184,E2 1338.184} C_VEL
LIN {X 0,Y 738.961,Z 1286.339,A -85,B 0,C 180,E1 1342.656,E2 1342.656} C_VEL
LIN {X 0,Y 739.338,Z 1297.82,A -85,B 0,C 180,E1 1347.088,E2 1347.088} C_VEL
LIN {X 0,Y 739.616,Z 1299.131,A -85,B 0,C 180,E1 1351.792,E2 1351.792} C_VEL
LIN {X 0,Y 739.599,Z 1287.258,A -85,B 0,C 180,E1 1357.1,E2 1357.1} C_VEL
LIN {X 0,Y 739.669,Z 1259.475,A -85,B 0,C 180,E1 1362.468,E2 1362.468} C_VEL
LIN {X 0,Y 740.037,Z 1218.878,A -85,B 0,C 180,E1 1367.171,E2 1367.171} C_VEL
LIN {X 0,Y 740.733,Z 1166.632,A -85,B 0,C 180,E1 1371.165,E2 1371.165} C_VEL
LIN {X 0,Y 741.503,Z 1106.518,A -85,B 0,C 180,E1 1374.17,E2 1374.17} C_VEL
LIN {X 0,Y 742.075,Z 1039.449,A -85,B 0,C 180,E1 1376.11,E2 1376.11} C_VEL
LIN {X 0,Y 740.122,Z 951.753,A -85,B 0,C 180,E1 1377.273,E2 1377.273} C_VEL
LIN {X 0,Y 739.588,Z 948.94,A -85,B 0,C 180,E1 1377.522,E2 1377.522} C_VEL
LIN {X 0,Y 739.122,Z 948.94,A -85,B 0,C 180,E1 1387.307,E2 1387.307} C_VEL
LIN {X 0,Y 738.778,Z 948.94,A -85,B 0,C 180,E1 1396.524,E2 1396.524} C_VEL
LIN {X 0,Y 739.081,Z 948.94,A -85,B 0,C 180,E1 1404.233,E2 1404.233} C_VEL
LIN {X 0,Y 739.566,Z 950.302,A -85,B 0,C 180,E1 1410.422,E2 1410.422} C_VEL
LIN {X 0,Y 741.687,Z 1016.977,A -85,B 0,C 180,E1 1412.086,E2 1412.086} C_VEL
LIN {X 0,Y 740.941,Z 1079.188,A -85,B 0,C 180,E1 1414.769,E2 1414.769} C_VEL
LIN {X 0,Y 740.173,Z 1134.536,A -85,B 0,C 180,E1 1418.51,E2 1418.51} C_VEL
LIN {X 0,Y 739.664,Z 1178.569,A -85,B 0,C 180,E1 1423.01,E2 1423.01} C_VEL
LIN {X 0,Y 739.245,Z 1208.942,A -85,B 0,C 180,E1 1427.863,E2 1427.863} C_VEL
LIN {X 0,Y 739.044,Z 1225.896,A -85,B 0,C 180,E1 1432.933,E2 1432.933} C_VEL
LIN {X 0,Y 738.707,Z 1229.979,A -85,B 0,C 180,E1 1437.067,E2 1437.067} C_VEL
LIN {X 0,Y 738.913,Z 1225.462,A -85,B 0,C 180,E1 1441.189,E2 1441.189} C_VEL
LIN {X 0,Y 739.212,Z 1208.231,A -85,B 0,C 180,E1 1446.2,E2 1446.2} C_VEL
LIN {X 0,Y 739.394,Z 1176.955,A -85,B 0,C 180,E1 1451.107,E2 1451.107} C_VEL
LIN {X 0,Y 740.076,Z 1132.675,A -85,B 0,C 180,E1 1455.553,E2 1455.553} C_VEL
LIN {X 0,Y 740.958,Z 1076.681,A -85,B 0,C 180,E1 1459.278,E2 1459.278} C_VEL
LIN {X 0,Y 741.733,Z 1012.611,A -85,B 0,C 180,E1 1461.968,E2 1461.968} C_VEL
LIN {X 0,Y 739.322,Z 948.94,A -85,B 0,C 180,E1 1463.611,E2 1463.611} C_VEL
LIN {X 0,Y 738.45,Z 948.94,A -85,B 0,C 180,E1 1470.25,E2 1470.25} C_VEL
LIN {X 0,Y 738.758,Z 948.94,A -85,B 0,C 180,E1 1477.7,E2 1477.7} C_VEL
LIN {X 0,Y 738.718,Z 948.94,A -85,B 0,C 180,E1 1486.483,E2 1486.483} C_VEL
LIN {X 0,Y 738.735,Z 948.94,A -85,B 0,C 180,E1 1494.269,E2 1494.269} C_VEL
LIN {X 0,Y 739.039,Z 948.94,A -85,B 0,C 180,E1 1501.121,E2 1501.121} C_VEL
LIN {X 0,Y 739.003,Z 948.94,A -85,B 0,C 180,E1 1509.18,E2 1509.18} C_VEL
LIN {X 0,Y 739.072,Z 949.007,A -85,B 0,C 180,E1 1514.58,E2 1514.58} C_VEL
LIN {X 0,Y 740.436,Z 1025.791,A -85,B 0,C 180,E1 1515.622,E2 1515.622} C_VEL
LIN {X 0,Y 740.099,Z 1072.811,A -85,B 0,C 180,E1 1517.463,E2 1517.463} C_VEL
LIN {X 0,Y 739.639,Z 1111.026,A -85,B 0,C 180,E1 1520.273,E2 1520.273} C_VEL
LIN {X 0,Y 739.409,Z 1137.145,A -85,B 0,C 180,E1 1523.786,E2 1523.786} C_VEL
LIN {X 0,Y 739.683,Z 1148.261,A -85,B 0,C 180,E1 1527.031,E2 1527.031} C_VEL
LIN {X 0,Y 739.638,Z 1147.719,A -85,B 0,C 180,E1 1531.146,E2 1531.146} C_VEL
LIN {X 0,Y 739.714,Z 1132.374,A -85,B 0,C 180,E1 1534.972,E2 1534.972} C_VEL
LIN {X 0,Y 739.924,Z 1102.992,A -85,B 0,C 180,E1 1538.372,E2 1538.372} C_VEL
LIN {X 0,Y 740.243,Z 1062.458,A -85,B 0,C 180,E1 1540.974,E2 1540.974} C_VEL
LIN {X 0,Y 740.5,Z 1014.153,A -85,B 0,C 180,E1 1542.552,E2 1542.552} C_VEL
LIN {X 0,Y 739.593,Z 948.94,A -85,B 0,C 180,E1 1543.354,E2 1543.354} C_VEL
LIN {X 0,Y 739.043,Z 948.94,A -85,B 0,C 180,E1 1551.025,E2 1551.025} C_VEL
LIN {X 0,Y 738.978,Z 948.94,A -85,B 0,C 180,E1 1559.177,E2 1559.177} C_VEL
LIN {X 0,Y 738.778,Z 948.94,A -85,B 0,C 180,E1 1567.704,E2 1567.704} C_VEL
LIN {X 0,Y 738.734,Z 948.94,A -85,B 0,C 180,E1 1576.489,E2 1576.489} C_VEL
LIN {X 0,Y 738.768,Z 948.94,A -85,B 0,C 180,E1 1584.168,E2 1584.168} C_VEL
LIN {X 0,Y 739.039,Z 948.94,A -85,B 0,C 180,E1 1591.129,E2 1591.129} C_VEL
LIN {X 0,Y 739.014,Z 948.94,A -85,B 0,C 180,E1 1599.011,E2 1599.011} C_VEL
LIN {X 0,Y 739.363,Z 948.94,A -85,B 0,C 180,E1 1607.54,E2 1607.54} C_VEL
LIN {X 0,Y 739.739,Z 948.94,A -85,B 0,C 180,E1 1617.048,E2 1617.048} C_VEL
LIN {X 0,Y 739.31,Z 948.94,A -85,B 0,C 180,E1 1624.655,E2 1624.655} C_VEL
LIN {X 0,Y 730.343,Z 948.94,A -85,B 0,C 180,E1 1627.333,E2 1627.333} C_VEL
LIN {X 0,Y 730.729,Z 948.94,A -85,B 0,C 180,E1 1633.808,E2 1633.808} C_VEL
LIN {X 0,Y 730.833,Z 948.94,A -85,B 0,C 180,E1 1641.299,E2 1641.299} C_VEL
LIN {X 0,Y 731.173,Z 948.94,A -85,B 0,C 180,E1 1649.184,E2 1649.184} C_VEL
LIN {X 0,Y 730.674,Z 948.94,A -85,B 0,C 180,E1 1656.97,E2 1656.97} C_VEL
LIN {X 0,Y 730.484,Z 948.94,A -85,B 0,C 180,E1 1664.269,E2 1664.269} C_VEL
LIN {X 0,Y 730.846,Z 948.94,A -85,B 0,C 180,E1 1672.272,E2 1672.272} C_VEL
LIN {X 0,Y 730.981,Z 948.94,A -85,B 0,C 180,E1 1678.077,E2 1678.077} C_VEL
LIN {X 0,Y 731.339,Z 950.589,A -85,B 0,C 180,E1 1682.359,E2 1682.359} C_VEL
LIN {X 0,Y 734.882,Z 967.029,A -85,B 0,C 180,E1 1682.681,E2 1682.681} C_VEL
LIN {X 0,Y 734.766,Z 1053.427,A -85,B 0,C 180,E1 1683.913,E2 1683.913} C_VEL
LIN {X 0,Y 733.879,Z 1119.736,A -85,B 0,C 180,E1 1686.121,E2 1686.121} C_VEL
LIN {X 0,Y 732.7,Z 1179.129,A -85,B 0,C 180,E1 1689.42,E2 1689.42} C_VEL
LIN {X 0,Y 731.861,Z 1227.358,A -85,B 0,C 180,E1 1693.468,E2 1693.468} C_VEL
LIN {X 0,Y 731.202,Z 1263.798,A -85,B 0,C 180,E1 1698.054,E2 1698.054} C_VEL
LIN {X 0,Y 731.022,Z 1286.34,A -85,B 0,C 180,E1 1702.576,E2 1702.576} C_VEL
LIN {X 0,Y 731.348,Z 1297.823,A -85,B 0,C 180,E1 1707.056,E2 1707.056} C_VEL
LIN {X 0,Y 731.619,Z 1299.133,A -85,B 0,C 180,E1 1711.812,E2 1711.812} C_VEL
LIN {X 0,Y 731.578,Z 1287.257,A -85,B 0,C 180,E1 1717.178,E2 1717.178} C_VEL
LIN {X 0,Y 731.678,Z 1259.479,A -85,B 0,C 180,E1 1722.606,E2 1722.606} C_VEL
LIN {X 0,Y 732.204,Z 1218.883,A -85,B 0,C 180,E1 1727.361,E2 1727.361} C_VEL
LIN {X 0,Y 733.095,Z 1167.109,A -85,B 0,C 180,E1 1731.367,E2 1731.367} C_VEL
LIN {X 0,Y 734.117,Z 1105.953,A -85,B 0,C 180,E1 1734.451,E2 1734.451} C_VEL
LIN {X 0,Y 734.878,Z 1039.47,A -85,B 0,C 180,E1 1736.386,E2 1736.386} C_VEL
LIN {X 0,Y 733.201,Z 954.161,A -85,B 0,C 180,E1 1737.526,E2 1737.526} C_VEL
LIN {X 0,Y 731.56,Z 948.94,A -85,B 0,C 180,E1 1737.734,E2 1737.734} C_VEL
LIN {X 0,Y 731.043,Z 948.94,A -85,B 0,C 180,E1 1747.791,E2 1747.791} C_VEL
LIN {X 0,Y 730.977,Z 948.94,A -85,B 0,C 180,E1 1755.942,E2 1755.942} C_VEL
LIN {X 0,Y 731.015,Z 948.94,A -85,B 0,C 180,E1 1763.734,E2 1763.734} C_VEL
LIN {X 0,Y 731.314,Z 950.258,A -85,B 0,C 180,E1 1770.098,E2 1770.098} C_VEL
LIN {X 0,Y 734.593,Z 998.509,A -85,B 0,C 180,E1 1771.256,E2 1771.256} C_VEL
LIN {X 0,Y 733.555,Z 1063.202,A -85,B 0,C 180,E1 1773.695,E2 1773.695} C_VEL
LIN {X 0,Y 732.426,Z 1121.59,A -85,B 0,C 180,E1 1777.273,E2 1777.273} C_VEL
LIN {X 0,Y 731.584,Z 1167.952,A -85,B 0,C 180,E1 1781.568,E2 1781.568} C_VEL
LIN {X 0,Y 731.074,Z 1200.911,A -85,B 0,C 180,E1 1786.199,E2 1786.199} C_VEL
LIN {X 0,Y 731.074,Z 1219.715,A -85,B 0,C 180,E1 1790.513,E2 1790.513} C_VEL
LIN {X 0,Y 731.579,Z 1228.69,A -85,B 0,C 180,E1 1794.655,E2 1794.655} C_VEL
LIN {X 0,Y 731.619,Z 1228.505,A -85,B 0,C 180,E1 1799.417,E2 1799.417} C_VEL
LIN {X 0,Y 731.756,Z 1213.731,A -85,B 0,C 180,E1 1805.051,E2 1805.051} C_VEL
LIN {X 0,Y 731.755,Z 1184.104,A -85,B 0,C 180,E1 1810.317,E2 1810.317} C_VEL
LIN {X 0,Y 732.336,Z 1141.121,A -85,B 0,C 180,E1 1815.027,E2 1815.027} C_VEL
LIN {X 0,Y 733.295,Z 1088.641,A -85,B 0,C 180,E1 1818.84,E2 1818.84} C_VEL
LIN {X 0,Y 734.151,Z 1026.188,A -85,B 0,C 180,E1 1821.777,E2 1821.777} C_VEL
LIN {X 0,Y 733.773,Z 957.409,A -85,B 0,C 180,E1 1823.601,E2 1823.601} C_VEL
LIN {X 0,Y 731.279,Z 948.94,A -85,B 0,C 180,E1 1823.887,E2 1823.887} C_VEL
LIN {X 0,Y 730.305,Z 948.94,A -85,B 0,C 180,E1 1830.623,E2 1830.623} C_VEL
LIN {X 0,Y 730.706,Z 948.94,A -85,B 0,C 180,E1 1837.805,E2 1837.805} C_VEL
LIN {X 0,Y 730.93,Z 948.94,A -85,B 0,C 180,E1 1845.901,E2 1845.901} C_VEL
LIN {X 0,Y 730.861,Z 948.94,A -85,B 0,C 180,E1 1853.689,E2 1853.689} C_VEL
LIN {X 0,Y 730.653,Z 948.94,A -85,B 0,C 180,E1 1862.112,E2 1862.112} C_VEL
LIN {X 0,Y 731.112,Z 948.94,A -85,B 0,C 180,E1 1868.673,E2 1868.673} C_VEL
LIN {X 0,Y 731.274,Z 950.167,A -85,B 0,C 180,E1 1874.435,E2 1874.435} C_VEL
LIN {X 0,Y 732.629,Z 1025.356,A -85,B 0,C 180,E1 1875.465,E2 1875.465} C_VEL
LIN {X 0,Y 732.228,Z 1072.933,A -85,B 0,C 180,E1 1877.344,E2 1877.344} C_VEL
LIN {X 0,Y 731.765,Z 1110.511,A -85,B 0,C 180,E1 1880.126,E2 1880.126} C_VEL
LIN {X 0,Y 731.45,Z 1137.087,A -85,B 0,C 180,E1 1883.718,E2 1883.718} C_VEL
LIN {X 0,Y 731.685,Z 1148.238,A -85,B 0,C 180,E1 1886.999,E2 1886.999} C_VEL
LIN {X 0,Y 731.644,Z 1147.742,A -85,B 0,C 180,E1 1891.159,E2 1891.159} C_VEL
LIN {X 0,Y 731.722,Z 1132.547,A -85,B 0,C 180,E1 1895.008,E2 1895.008} C_VEL
LIN {X 0,Y 731.97,Z 1103.13,A -85,B 0,C 180,E1 1898.463,E2 1898.463} C_VEL
LIN {X 0,Y 732.389,Z 1062.699,A -85,B 0,C 180,E1 1901.094,E2 1901.094} C_VEL
LIN {X 0,Y 732.718,Z 1014.748,A -85,B 0,C 180,E1 1902.688,E2 1902.688} C_VEL
LIN {X 0,Y 731.429,Z 948.94,A -85,B 0,C 180,E1 1903.616,E2 1903.616} C_VEL
LIN {X 0,Y 730.863,Z 948.94,A -85,B 0,C 180,E1 1911.271,E2 1911.271} C_VEL
LIN {X 0,Y 730.98,Z 948.94,A -85,B 0,C 180,E1 1919.161,E2 1919.161} C_VEL
LIN {X 0,Y 730.763,Z 948.94,A -85,B 0,C 180,E1 1927.733,E2 1927.733} C_VEL
LIN {X 0,Y 730.934,Z 948.94,A -85,B 0,C 180,E1 1935.906,E2 1935.906} C_VEL
LIN {X 0,Y 730.842,Z 948.94,A -85,B 0,C 180,E1 1943.695,E2 1943.695} C_VEL
LIN {X 0,Y 730.655,Z 948.94,A -85,B 0,C 180,E1 1952.121,E2 1952.121} C_VEL
LIN {X 0,Y 731.067,Z 948.94,A -85,B 0,C 180,E1 1958.683,E2 1958.683} C_VEL
LIN {X 0,Y 731.381,Z 948.94,A -85,B 0,C 180,E1 1967.402,E2 1967.402} C_VEL
LIN {X 0,Y 731.725,Z 948.94,A -85,B 0,C 180,E1 1977.016,E2 1977.016} C_VEL
LIN {X 0,Y 731.306,Z 948.94,A -85,B 0,C 180,E1 1985.347,E2 1985.347} C_VEL
LIN {X 0,Y 730.343,Z 948.94,A -85,B 0,C 180,E1 1987.333,E2 1987.333} C_VEL
LIN {X 0,Y 722.488,Z 948.94,A -85,B 0,C 180,E1 1990.066,E2 1990.066} C_VEL
LIN {X 0,Y 722.23,Z 948.94,A -85,B 0,C 180,E1 1995.218,E2 1995.218} C_VEL
LIN {X 0,Y 722.682,Z 948.94,A -85,B 0,C 180,E1 2001.551,E2 2001.551} C_VEL
LIN {X 0,Y 723.012,Z 948.94,A -85,B 0,C 180,E1 2009.546,E2 2009.546} C_VEL
LIN {X 0,Y 722.747,Z 948.94,A -85,B 0,C 180,E1 2016.749,E2 2016.749} C_VEL
LIN {X 0,Y 722.711,Z 948.94,A -85,B 0,C 180,E1 2023.633,E2 2023.633} C_VEL
LIN {X 0,Y 722.936,Z 948.94,A -85,B 0,C 180,E1 2031.916,E2 2031.916} C_VEL
LIN {X 0,Y 722.699,Z 948.94,A -85,B 0,C 180,E1 2039.08,E2 2039.08} C_VEL
LIN {X 0,Y 723.242,Z 950.854,A -85,B 0,C 180,E1 2042.026,E2 2042.026} C_VEL
LIN {X 0,Y 727.771,Z 967.247,A -85,B 0,C 180,E1 2042.394,E2 2042.394} C_VEL
LIN {X 0,Y 727.551,Z 1053.044,A -85,B 0,C 180,E1 2043.625,E2 2043.625} C_VEL
LIN {X 0,Y 726.463,Z 1118.378,A -85,B 0,C 180,E1 2045.802,E2 2045.802} C_VEL
LIN {X 0,Y 725.111,Z 1178.169,A -85,B 0,C 180,E1 2049.126,E2 2049.126} C_VEL
LIN {X 0,Y 724.023,Z 1227.432,A -85,B 0,C 180,E1 2053.291,E2 2053.291} C_VEL
LIN {X 0,Y 723.267,Z 1263.801,A -85,B 0,C 180,E1 2057.921,E2 2057.921} C_VEL
LIN {X 0,Y 722.933,Z 1287.491,A -85,B 0,C 180,E1 2062.796,E2 2062.796} C_VEL
LIN {X 0,Y 723.36,Z 1297.827,A -85,B 0,C 180,E1 2067.024,E2 2067.024} C_VEL
LIN {X 0,Y 723.596,Z 1299.135,A -85,B 0,C 180,E1 2071.832,E2 2071.832} C_VEL
LIN {X 0,Y 723.541,Z 1287.256,A -85,B 0,C 180,E1 2077.258,E2 2077.258} C_VEL
LIN {X 0,Y 723.8,Z 1261.45,A -85,B 0,C 180,E1 2082.438,E2 2082.438} C_VEL
LIN {X 0,Y 724.369,Z 1221.395,A -85,B 0,C 180,E1 2087.31,E2 2087.31} C_VEL
LIN {X 0,Y 725.432,Z 1169.803,A -85,B 0,C 180,E1 2091.431,E2 2091.431} C_VEL
LIN {X 0,Y 726.692,Z 1108.964,A -85,B 0,C 180,E1 2094.598,E2 2094.598} C_VEL
LIN {X 0,Y 727.655,Z 1042.905,A -85,B 0,C 180,E1 2096.596,E2 2096.596} C_VEL
LIN {X 0,Y 725.904,Z 956.122,A -85,B 0,C 180,E1 2097.805,E2 2097.805} C_VEL
LIN {X 0,Y 723.509,Z 948.94,A -85,B 0,C 180,E1 2098.033,E2 2098.033} C_VEL
LIN {X 0,Y 722.881,Z 948.94,A -85,B 0,C 180,E1 2108.294,E2 2108.294} C_VEL
LIN {X 0,Y 722.697,Z 948.94,A -85,B 0,C 180,E1 2116.455,E2 2116.455} C_VEL
LIN {X 0,Y 722.785,Z 948.94,A -85,B 0,C 180,E1 2124.741,E2 2124.741} C_VEL
LIN {X 0,Y 723.084,Z 949.831,A -85,B 0,C 180,E1 2129.762,E2 2129.762} C_VEL
LIN {X 0,Y 727.269,Z 973.151,A -85,B 0,C 180,E1 2130.349,E2 2130.349} C_VEL
LIN {X 0,Y 726.601,Z 1039.743,A -85,B 0,C 180,E1 2132.386,E2 2132.386} C_VEL
LIN {X 0,Y 725.43,Z 1100.181,A -85,B 0,C 180,E1 2135.552,E2 2135.552} C_VEL
LIN {X 0,Y 724.547,Z 1151.542,A -85,B 0,C 180,E1 2139.667,E2 2139.667} C_VEL
LIN {X 0,Y 723.926,Z 1190.561,A -85,B 0,C 180,E1 2144.383,E2 2144.383} C_VEL
LIN {X 0,Y 723.484,Z 1217.433,A -85,B 0,C 180,E1 2149.74,E2 2149.74} C_VEL
LIN {X 0,Y 723.576,Z 1228.651,A -85,B 0,C 180,E1 2154.595,E2 2154.595} C_VEL
LIN {X 0,Y 723.609,Z 1228.539,A -85,B 0,C 180,E1 2159.411,E2 2159.411} C_VEL
LIN {X 0,Y 723.803,Z 1214.371,A -85,B 0,C 180,E1 2164.976,E2 2164.976} C_VEL
LIN {X 0,Y 723.846,Z 1185.439,A -85,B 0,C 180,E1 2170.279,E2 2170.279} C_VEL
LIN {X 0,Y 724.521,Z 1143.257,A -85,B 0,C 180,E1 2175.037,E2 2175.037} C_VEL
LIN {X 0,Y 725.691,Z 1089.642,A -85,B 0,C 180,E1 2179.023,E2 2179.023} C_VEL
LIN {X 0,Y 726.79,Z 1027.667,A -85,B 0,C 180,E1 2181.988,E2 2181.988} C_VEL
LIN {X 0,Y 726.647,Z 959.172,A -85,B 0,C 180,E1 2183.853,E2 2183.853} C_VEL
LIN {X 0,Y 723.218,Z 948.94,A -85,B 0,C 180,E1 2184.17,E2 2184.17} C_VEL
LIN {X 0,Y 722.165,Z 948.94,A -85,B 0,C 180,E1 2191.006,E2 2191.006} C_VEL
LIN {X 0,Y 722.465,Z 948.94,A -85,B 0,C 180,E1 2198.313,E2 2198.313} C_VEL
LIN {X 0,Y 722.652,Z 948.94,A -85,B 0,C 180,E1 2206.454,E2 2206.454} C_VEL
LIN {X 0,Y 722.737,Z 948.94,A -85,B 0,C 180,E1 2213.973,E2 2213.973} C_VEL
LIN {X 0,Y 722.758,Z 948.94,A -85,B 0,C 180,E1 2221.78,E2 2221.78} C_VEL
LIN {X 0,Y 722.765,Z 948.94,A -85,B 0,C 180,E1 2229.703,E2 2229.703} C_VEL
LIN {X 0,Y 723.408,Z 950.3,A -85,B 0,C 180,E1 2234.275,E2 2234.275} C_VEL
LIN {X 0,Y 724.868,Z 1024.881,A -85,B 0,C 180,E1 2235.306,E2 2235.306} C_VEL
LIN {X 0,Y 724.415,Z 1071.758,A -85,B 0,C 180,E1 2237.152,E2 2237.152} C_VEL
LIN {X 0,Y 723.828,Z 1110.546,A -85,B 0,C 180,E1 2240.032,E2 2240.032} C_VEL
LIN {X 0,Y 723.481,Z 1137.028,A -85,B 0,C 180,E1 2243.649,E2 2243.649} C_VEL
LIN {X 0,Y 723.685,Z 1148.216,A -85,B 0,C 180,E1 2246.966,E2 2246.966} C_VEL
LIN {X 0,Y 723.638,Z 1147.765,A -85,B 0,C 180,E1 2251.172,E2 2251.172} C_VEL
LIN {X 0,Y 723.67,Z 1132.101,A -85,B 0,C 180,E1 2255.153,E2 2255.153} C_VEL
LIN {X 0,Y 724,Z 1103.265,A -85,B 0,C 180,E1 2258.557,E2 2258.557} C_VEL
LIN {X 0,Y 724.524,Z 1062.939,A -85,B 0,C 180,E1 2261.216,E2 2261.216} C_VEL
LIN {X 0,Y 724.936,Z 1014.945,A -85,B 0,C 180,E1 2262.834,E2 2262.834} C_VEL
LIN {X 0,Y 723.363,Z 948.94,A -85,B 0,C 180,E1 2263.703,E2 2263.703} C_VEL
LIN {X 0,Y 722.713,Z 948.94,A -85,B 0,C 180,E1 2271.523,E2 2271.523} C_VEL
LIN {X 0,Y 722.783,Z 948.94,A -85,B 0,C 180,E1 2279.524,E2 2279.524} C_VEL
LIN {X 0,Y 722.515,Z 948.94,A -85,B 0,C 180,E1 2288.241,E2 2288.241} C_VEL
LIN {X 0,Y 722.737,Z 948.94,A -85,B 0,C 180,E1 2296.365,E2 2296.365} C_VEL
LIN {X 0,Y 722.757,Z 948.94,A -85,B 0,C 180,E1 2303.872,E2 2303.872} C_VEL
LIN {X 0,Y 722.778,Z 948.94,A -85,B 0,C 180,E1 2311.791,E2 2311.791} C_VEL
LIN {X 0,Y 722.627,Z 948.94,A -85,B 0,C 180,E1 2319.71,E2 2319.71} C_VEL
LIN {X 0,Y 723.368,Z 948.94,A -85,B 0,C 180,E1 2327.26,E2 2327.26} C_VEL
LIN {X 0,Y 723.684,Z 948.94,A -85,B 0,C 180,E1 2336.983,E2 2336.983} C_VEL
LIN {X 0,Y 723.271,Z 948.94,A -85,B 0,C 180,E1 2345.407,E2 2345.407} C_VEL
LIN {X 0,Y 722.488,Z 948.94,A -85,B 0,C 180,E1 2350.066,E2 2350.066} C_VEL
LIN {X 0,Y 715.237,Z 948.94,A -85,B 0,C 180,E1 2352.844,E2 2352.844} C_VEL
LIN {X 0,Y 714.535,Z 948.94,A -85,B 0,C 180,E1 2361.81,E2 2361.81} C_VEL
LIN {X 0,Y 714.87,Z 948.94,A -85,B 0,C 180,E1 2369.917,E2 2369.917} C_VEL
LIN {X 0,Y 714.6,Z 948.94,A -85,B 0,C 180,E1 2377.279,E2 2377.279} C_VEL
LIN {X 0,Y 714.708,Z 948.94,A -85,B 0,C 180,E1 2383.629,E2 2383.629} C_VEL
LIN {X 0,Y 714.962,Z 948.94,A -85,B 0,C 180,E1 2391.28,E2 2391.28} C_VEL
LIN {X 0,Y 714.793,Z 948.94,A -85,B 0,C 180,E1 2398.699,E2 2398.699} C_VEL
LIN {X 0,Y 715.079,Z 950.577,A -85,B 0,C 180,E1 2401.675,E2 2401.675} C_VEL
LIN {X 0,Y 720.694,Z 968.217,A -85,B 0,C 180,E1 2402.11,E2 2402.11} C_VEL
LIN {X 0,Y 720.332,Z 1053.657,A -85,B 0,C 180,E1 2403.355,E2 2403.355} C_VEL
LIN {X 0,Y 719.024,Z 1119.888,A -85,B 0,C 180,E1 2405.602,E2 2405.602} C_VEL
LIN {X 0,Y 717.435,Z 1179.297,A -85,B 0,C 180,E1 2408.972,E2 2408.972} C_VEL
LIN {X 0,Y 716.141,Z 1229.019,A -85,B 0,C 180,E1 2413.272,E2 2413.272} C_VEL
LIN {X 0,Y 715.343,Z 1263.952,A -85,B 0,C 180,E1 2417.809,E2 2417.809} C_VEL
LIN {X 0,Y 714.964,Z 1287.492,A -85,B 0,C 180,E1 2422.715,E2 2422.715} C_VEL
LIN {X 0,Y 715.389,Z 1297.83,A -85,B 0,C 180,E1 2426.991,E2 2426.991} C_VEL
LIN {X 0,Y 715.572,Z 1299.138,A -85,B 0,C 180,E1 2431.853,E2 2431.853} C_VEL
LIN {X 0,Y 715.514,Z 1287.256,A -85,B 0,C 180,E1 2437.34,E2 2437.34} C_VEL
LIN {X 0,Y 715.732,Z 1260.503,A -85,B 0,C 180,E1 2442.731,E2 2442.731} C_VEL
LIN {X 0,Y 716.503,Z 1220.982,A -85,B 0,C 180,E1 2447.547,E2 2447.547} C_VEL
LIN {X 0,Y 717.844,Z 1168.701,A -85,B 0,C 180,E1 2451.741,E2 2451.741} C_VEL
LIN {X 0,Y 719.373,Z 1107.868,A -85,B 0,C 180,E1 2454.91,E2 2454.91} C_VEL
LIN {X 0,Y 720.476,Z 1041.979,A -85,B 0,C 180,E1 2456.902,E2 2456.902} C_VEL
LIN {X 0,Y 718.828,Z 958.205,A -85,B 0,C 180,E1 2458.08,E2 2458.08} C_VEL
LIN {X 0,Y 715.475,Z 948.94,A -85,B 0,C 180,E1 2458.337,E2 2458.337} C_VEL
LIN {X 0,Y 714.916,Z 948.94,A -85,B 0,C 180,E1 2467.256,E2 2467.256} C_VEL
LIN {X 0,Y 714.737,Z 948.94,A -85,B 0,C 180,E1 2476.373,E2 2476.373} C_VEL
LIN {X 0,Y 714.743,Z 948.94,A -85,B 0,C 180,E1 2484.866,E2 2484.866} C_VEL
LIN {X 0,Y 715.07,Z 950.786,A -85,B 0,C 180,E1 2489.446,E2 2489.446} C_VEL
LIN {X 0,Y 720.016,Z 971.329,A -85,B 0,C 180,E1 2490.02,E2 2490.02} C_VEL
LIN {X 0,Y 719.238,Z 1038.926,A -85,B 0,C 180,E1 2492.085,E2 2492.085} C_VEL
LIN {X 0,Y 717.839,Z 1099.591,A -85,B 0,C 180,E1 2495.276,E2 2495.276} C_VEL
LIN {X 0,Y 716.718,Z 1151.301,A -85,B 0,C 180,E1 2499.448,E2 2499.448} C_VEL
LIN {X 0,Y 715.99,Z 1191.126,A -85,B 0,C 180,E1 2504.331,E2 2504.331} C_VEL
LIN {X 0,Y 715.578,Z 1217.305,A -85,B 0,C 180,E1 2509.625,E2 2509.625} C_VEL
LIN {X 0,Y 715.553,Z 1228.611,A -85,B 0,C 180,E1 2514.535,E2 2514.535} C_VEL
LIN {X 0,Y 715.611,Z 1228.571,A -85,B 0,C 180,E1 2519.404,E2 2519.404} C_VEL
LIN {X 0,Y 715.779,Z 1214.504,A -85,B 0,C 180,E1 2525.031,E2 2525.031} C_VEL
LIN {X 0,Y 715.887,Z 1185.691,A -85,B 0,C 180,E1 2530.394,E2 2530.394} C_VEL
LIN {X 0,Y 716.699,Z 1143.66,A -85,B 0,C 180,E1 2535.205,E2 2535.205} C_VEL
LIN {X 0,Y 718.101,Z 1090.266,A -85,B 0,C 180,E1 2539.228,E2 2539.228} C_VEL
LIN {X 0,Y 719.441,Z 1029.021,A -85,B 0,C 180,E1 2542.209,E2 2542.209} C_VEL
LIN {X 0,Y 719.092,Z 960.236,A -85,B 0,C 180,E1 2544.14,E2 2544.14} C_VEL
LIN {X 0,Y 715.132,Z 948.94,A -85,B 0,C 180,E1 2544.595,E2 2544.595} C_VEL
LIN {X 0,Y 714.087,Z 948.94,A -85,B 0,C 180,E1 2551.397,E2 2551.397} C_VEL
LIN {X 0,Y 714.778,Z 948.94,A -85,B 0,C 180,E1 2557.257,E2 2557.257} C_VEL
LIN {X 0,Y 714.677,Z 948.94,A -85,B 0,C 180,E1 2566.33,E2 2566.33} C_VEL
LIN {X 0,Y 714.634,Z 948.94,A -85,B 0,C 180,E1 2574.24,E2 2574.24} C_VEL
LIN {X 0,Y 714.748,Z 948.94,A -85,B 0,C 180,E1 2581.822,E2 2581.822} C_VEL
LIN {X 0,Y 714.827,Z 948.94,A -85,B 0,C 180,E1 2589.467,E2 2589.467} C_VEL
LIN {X 0,Y 715.426,Z 950.513,A -85,B 0,C 180,E1 2594.109,E2 2594.109} C_VEL
LIN {X 0,Y 717.08,Z 1025.92,A -85,B 0,C 180,E1 2595.182,E2 2595.182} C_VEL
LIN {X 0,Y 716.542,Z 1072.566,A -85,B 0,C 180,E1 2597.066,E2 2597.066} C_VEL
LIN {X 0,Y 715.942,Z 1110.104,A -85,B 0,C 180,E1 2599.889,E2 2599.889} C_VEL
LIN {X 0,Y 715.518,Z 1136.97,A -85,B 0,C 180,E1 2603.578,E2 2603.578} C_VEL
LIN {X 0,Y 715.702,Z 1148.193,A -85,B 0,C 180,E1 2606.932,E2 2606.932} C_VEL
LIN {X 0,Y 715.651,Z 1147.788,A -85,B 0,C 180,E1 2611.185,E2 2611.185} C_VEL
LIN {X 0,Y 715.655,Z 1132.171,A -85,B 0,C 180,E1 2615.211,E2 2615.211} C_VEL
LIN {X 0,Y 716.04,Z 1103.396,A -85,B 0,C 180,E1 2618.653,E2 2618.653} C_VEL
LIN {X 0,Y 716.676,Z 1063.177,A -85,B 0,C 180,E1 2621.34,E2 2621.34} C_VEL
LIN {X 0,Y 717.176,Z 1015.496,A -85,B 0,C 180,E1 2622.975,E2 2622.975} C_VEL
LIN {X 0,Y 715.245,Z 948.94,A -85,B 0,C 180,E1 2623.909,E2 2623.909} C_VEL
LIN {X 0,Y 714.559,Z 948.94,A -85,B 0,C 180,E1 2631.781,E2 2631.781} C_VEL
LIN {X 0,Y 714.582,Z 948.94,A -85,B 0,C 180,E1 2639.897,E2 2639.897} C_VEL
LIN {X 0,Y 714.771,Z 948.94,A -85,B 0,C 180,E1 2647.202,E2 2647.202} C_VEL
LIN {X 0,Y 714.747,Z 948.94,A -85,B 0,C 180,E1 2656.341,E2 2656.341} C_VEL
LIN {X 0,Y 714.482,Z 948.94,A -85,B 0,C 180,E1 2664.791,E2 2664.791} C_VEL
LIN {X 0,Y 714.789,Z 948.94,A -85,B 0,C 180,E1 2671.689,E2 2671.689} C_VEL
LIN {X 0,Y 714.72,Z 948.94,A -85,B 0,C 180,E1 2679.476,E2 2679.476} C_VEL
LIN {X 0,Y 715.389,Z 948.94,A -85,B 0,C 180,E1 2687.116,E2 2687.116} C_VEL
LIN {X 0,Y 715.643,Z 948.94,A -85,B 0,C 180,E1 2696.949,E2 2696.949} C_VEL
LIN {X 0,Y 715.22,Z 948.94,A -85,B 0,C 180,E1 2705.468,E2 2705.468} C_VEL
LIN {X 0,Y 715.237,Z 948.94,A -85,B 0,C 180,E1 2712.844,E2 2712.844} C_VEL
LIN {X 0,Y 706.161,Z 948.94,A -85,B 0,C 180,E1 2715.607,E2 2715.607} C_VEL
LIN {X 0,Y 706.42,Z 948.94,A -85,B 0,C 180,E1 2722.073,E2 2722.073} C_VEL
LIN {X 0,Y 706.784,Z 948.94,A -85,B 0,C 180,E1 2730.295,E2 2730.295} C_VEL
LIN {X 0,Y 706.517,Z 948.94,A -85,B 0,C 180,E1 2737.738,E2 2737.738} C_VEL
LIN {X 0,Y 706.453,Z 948.94,A -85,B 0,C 180,E1 2744.271,E2 2744.271} C_VEL
LIN {X 0,Y 706.774,Z 948.94,A -85,B 0,C 180,E1 2752.317,E2 2752.317} C_VEL
LIN {X 0,Y 706.627,Z 948.94,A -85,B 0,C 180,E1 2759.731,E2 2759.731} C_VEL
LIN {X 0,Y 706.978,Z 950.537,A -85,B 0,C 180,E1 2761.32,E2 2761.32} C_VEL
LIN {X 0,Y 713.643,Z 968.486,A -85,B 0,C 180,E1 2761.813,E2 2761.813} C_VEL
LIN {X 0,Y 713.159,Z 1054.057,A -85,B 0,C 180,E1 2763.076,E2 2763.076} C_VEL
LIN {X 0,Y 711.672,Z 1119.205,A -85,B 0,C 180,E1 2765.303,E2 2765.303} C_VEL
LIN {X 0,Y 709.815,Z 1178.862,A -85,B 0,C 180,E1 2768.704,E2 2768.704} C_VEL
LIN {X 0,Y 708.351,Z 1228.248,A -85,B 0,C 180,E1 2772.998,E2 2772.998} C_VEL
LIN {X 0,Y 707.371,Z 1264.907,A -85,B 0,C 180,E1 2777.827,E2 2777.827} C_VEL
LIN {X 0,Y 706.997,Z 1287.492,A -85,B 0,C 180,E1 2782.632,E2 2782.632} C_VEL
LIN {X 0,Y 707.4,Z 1297.834,A -85,B 0,C 180,E1 2786.957,E2 2786.957} C_VEL
LIN {X 0,Y 707.55,Z 1299.14,A -85,B 0,C 180,E1 2791.874,E2 2791.874} C_VEL
LIN {X 0,Y 707.476,Z 1287.255,A -85,B 0,C 180,E1 2797.424,E2 2797.424} C_VEL
LIN {X 0,Y 707.773,Z 1260.836,A -85,B 0,C 180,E1 2802.824,E2 2802.824} C_VEL
LIN {X 0,Y 708.686,Z 1220.455,A -85,B 0,C 180,E1 2807.8,E2 2807.8} C_VEL
LIN {X 0,Y 710.26,Z 1168.707,A -85,B 0,C 180,E1 2811.985,E2 2811.985} C_VEL
LIN {X 0,Y 712.029,Z 1107.972,A -85,B 0,C 180,E1 2815.181,E2 2815.181} C_VEL
LIN {X 0,Y 713.364,Z 1041.522,A -85,B 0,C 180,E1 2817.203,E2 2817.203} C_VEL
LIN {X 0,Y 711.771,Z 960.545,A -85,B 0,C 180,E1 2818.357,E2 2818.357} C_VEL
LIN {X 0,Y 707.352,Z 948.94,A -85,B 0,C 180,E1 2818.771,E2 2818.771} C_VEL
LIN {X 0,Y 706.65,Z 948.94,A -85,B 0,C 180,E1 2828.393,E2 2828.393} C_VEL
LIN {X 0,Y 706.802,Z 948.94,A -85,B 0,C 180,E1 2836.027,E2 2836.027} C_VEL
LIN {X 0,Y 706.6,Z 948.94,A -85,B 0,C 180,E1 2845.318,E2 2845.318} C_VEL
LIN {X 0,Y 706.96,Z 950.918,A -85,B 0,C 180,E1 2849.105,E2 2849.105} C_VEL
LIN {X 0,Y 712.849,Z 972.4,A -85,B 0,C 180,E1 2849.75,E2 2849.75} C_VEL
LIN {X 0,Y 711.871,Z 1039.559,A -85,B 0,C 180,E1 2851.836,E2 2851.836} C_VEL
LIN {X 0,Y 710.255,Z 1099.842,A -85,B 0,C 180,E1 2855.05,E2 2855.05} C_VEL
LIN {X 0,Y 708.9,Z 1150.418,A -85,B 0,C 180,E1 2859.16,E2 2859.16} C_VEL
LIN {X 0,Y 708.128,Z 1188.904,A -85,B 0,C 180,E1 2863.833,E2 2863.833} C_VEL
LIN {X 0,Y 707.752,Z 1216.019,A -85,B 0,C 180,E1 2869.197,E2 2869.197} C_VEL
LIN {X 0,Y 707.535,Z 1228.572,A -85,B 0,C 180,E1 2874.472,E2 2874.472} C_VEL
LIN {X 0,Y 707.6,Z 1228.603,A -85,B 0,C 180,E1 2879.398,E2 2879.398} C_VEL
LIN {X 0,Y 707.681,Z 1214.056,A -85,B 0,C 180,E1 2885.242,E2 2885.242} C_VEL
LIN {X 0,Y 707.88,Z 1184.859,A -85,B 0,C 180,E1 2890.669,E2 2890.669} C_VEL
LIN {X 0,Y 708.905,Z 1142.33,A -85,B 0,C 180,E1 2895.536,E2 2895.536} C_VEL
LIN {X 0,Y 710.592,Z 1088.985,A -85,B 0,C 180,E1 2899.558,E2 2899.558} C_VEL
LIN {X 0,Y 712.214,Z 1026.844,A -85,B 0,C 180,E1 2902.57,E2 2902.57} C_VEL
LIN {X 0,Y 711.357,Z 960.959,A -85,B 0,C 180,E1 2904.446,E2 2904.446} C_VEL
LIN {X 0,Y 707.108,Z 948.94,A -85,B 0,C 180,E1 2905.014,E2 2905.014} C_VEL
LIN {X 0,Y 706.036,Z 948.94,A -85,B 0,C 180,E1 2911.855,E2 2911.855} C_VEL
LIN {X 0,Y 706.365,Z 948.94,A -85,B 0,C 180,E1 2918.321,E2 2918.321} C_VEL
LIN {X 0,Y 706.744,Z 948.94,A -85,B 0,C 180,E1 2926.026,E2 2926.026} C_VEL
LIN {X 0,Y 706.692,Z 948.94,A -85,B 0,C 180,E1 2933.775,E2 2933.775} C_VEL
LIN {X 0,Y 706.829,Z 948.94,A -85,B 0,C 180,E1 2941.085,E2 2941.085} C_VEL
LIN {X 0,Y 706.85,Z 948.94,A -85,B 0,C 180,E1 2949.225,E2 2949.225} C_VEL
LIN {X 0,Y 707.427,Z 950.751,A -85,B 0,C 180,E1 2953.94,E2 2953.94} C_VEL
LIN {X 0,Y 709.323,Z 1024.524,A -85,B 0,C 180,E1 2954.992,E2 2954.992} C_VEL
LIN {X 0,Y 708.774,Z 1070.609,A -85,B 0,C 180,E1 2956.822,E2 2956.822} C_VEL
LIN {X 0,Y 708.106,Z 1108.521,A -85,B 0,C 180,E1 2959.631,E2 2959.631} C_VEL
LIN {X 0,Y 707.758,Z 1135.36,A -85,B 0,C 180,E1 2963.198,E2 2963.198} C_VEL
LIN {X 0,Y 707.698,Z 1148.171,A -85,B 0,C 180,E1 2966.897,E2 2966.897} C_VEL
LIN {X 0,Y 707.661,Z 1147.811,A -85,B 0,C 180,E1 2971.198,E2 2971.198} C_VEL
LIN {X 0,Y 707.689,Z 1132.649,A -85,B 0,C 180,E1 2975.198,E2 2975.198} C_VEL
LIN {X 0,Y 708.1,Z 1103.526,A -85,B 0,C 180,E1 2978.751,E2 2978.751} C_VEL
LIN {X 0,Y 708.849,Z 1063.415,A -85,B 0,C 180,E1 2981.467,E2 2981.467} C_VEL
LIN {X 0,Y 709.417,Z 1016.583,A -85,B 0,C 180,E1 2983.108,E2 2983.108} C_VEL
LIN {X 0,Y 707.154,Z 948.94,A -85,B 0,C 180,E1 2984.025,E2 2984.025} C_VEL
LIN {X 0,Y 706.441,Z 948.94,A -85,B 0,C 180,E1 2992.045,E2 2992.045} C_VEL
LIN {X 0,Y 706.412,Z 948.94,A -85,B 0,C 180,E1 3000.279,E2 3000.279} C_VEL
LIN {X 0,Y 706.36,Z 948.94,A -85,B 0,C 180,E1 3008.325,E2 3008.325} C_VEL
LIN {X 0,Y 706.842,Z 948.94,A -85,B 0,C 180,E1 3015.936,E2 3015.936} C_VEL
LIN {X 0,Y 706.672,Z 948.94,A -85,B 0,C 180,E1 3023.782,E2 3023.782} C_VEL
LIN {X 0,Y 706.823,Z 948.94,A -85,B 0,C 180,E1 3031.094,E2 3031.094} C_VEL
LIN {X 0,Y 706.754,Z 948.94,A -85,B 0,C 180,E1 3039.234,E2 3039.234} C_VEL
LIN {X 0,Y 707.381,Z 948.94,A -85,B 0,C 180,E1 3047.266,E2 3047.266} C_VEL
LIN {X 0,Y 707.598,Z 948.94,A -85,B 0,C 180,E1 3056.923,E2 3056.923} C_VEL
LIN {X 0,Y 707.19,Z 948.94,A -85,B 0,C 180,E1 3065.53,E2 3065.53} C_VEL
LIN {X 0,Y 707.151,Z 948.94,A -85,B 0,C 180,E1 3073.012,E2 3073.012} C_VEL
LIN {X 0,Y 706.161,Z 948.94,A -85,B 0,C 180,E1 3075.607,E2 3075.607} C_VEL
LIN {X 0,Y 698.545,Z 948.94,A -85,B 0,C 180,E1 3078.431,E2 3078.431} C_VEL
LIN {X 0,Y 698.371,Z 948.94,A -85,B 0,C 180,E1 3086.444,E2 3086.444} C_VEL
LIN {X 0,Y 698.913,Z 948.94,A -85,B 0,C 180,E1 3093.612,E2 3093.612} C_VEL
LIN {X 0,Y 698.89,Z 948.94,A -85,B 0,C 180,E1 3101.544,E2 3101.544} C_VEL
LIN {X 0,Y 698.982,Z 948.94,A -85,B 0,C 180,E1 3110.412,E2 3110.412} C_VEL
LIN {X 0,Y 698.91,Z 948.94,A -85,B 0,C 180,E1 3117.904,E2 3117.904} C_VEL
LIN {X 0,Y 698.954,Z 950.739,A -85,B 0,C 180,E1 3120.962,E2 3120.962} C_VEL
LIN {X 0,Y 706.619,Z 974.229,A -85,B 0,C 180,E1 3121.573,E2 3121.573} C_VEL
LIN {X 0,Y 705.988,Z 1055.199,A -85,B 0,C 180,E1 3122.809,E2 3122.809} C_VEL
LIN {X 0,Y 704.264,Z 1121.058,A -85,B 0,C 180,E1 3125.109,E2 3125.109} C_VEL
LIN {X 0,Y 702.154,Z 1180.848,A -85,B 0,C 180,E1 3128.604,E2 3128.604} C_VEL
LIN {X 0,Y 700.424,Z 1230.321,A -85,B 0,C 180,E1 3133.028,E2 3133.028} C_VEL
LIN {X 0,Y 699.359,Z 1266.46,A -85,B 0,C 180,E1 3137.945,E2 3137.945} C_VEL
LIN {X 0,Y 699.036,Z 1287.493,A -85,B 0,C 180,E1 3142.548,E2 3142.548} C_VEL
LIN {X 0,Y 699.415,Z 1297.837,A -85,B 0,C 180,E1 3146.922,E2 3146.922} C_VEL
LIN {X 0,Y 699.547,Z 1299.142,A -85,B 0,C 180,E1 3151.895,E2 3151.895} C_VEL
LIN {X 0,Y 699.436,Z 1287.255,A -85,B 0,C 180,E1 3157.51,E2 3157.51} C_VEL
LIN {X 0,Y 699.791,Z 1260.838,A -85,B 0,C 180,E1 3162.973,E2 3162.973} C_VEL
LIN {X 0,Y 700.855,Z 1221.898,A -85,B 0,C 180,E1 3167.861,E2 3167.861} C_VEL
LIN {X 0,Y 702.659,Z 1170.064,A -85,B 0,C 180,E1 3172.146,E2 3172.146} C_VEL
LIN {X 0,Y 704.635,Z 1109.626,A -85,B 0,C 180,E1 3175.392,E2 3175.392} C_VEL
LIN {X 0,Y 706.18,Z 1044.049,A -85,B 0,C 180,E1 3177.448,E2 3177.448} C_VEL
LIN {X 0,Y 704.746,Z 962.953,A -85,B 0,C 180,E1 3178.638,E2 3178.638} C_VEL
LIN {X 0,Y 699.26,Z 948.94,A -85,B 0,C 180,E1 3179.135,E2 3179.135} C_VEL
LIN {X 0,Y 698.665,Z 948.94,A -85,B 0,C 180,E1 3188.277,E2 3188.277} C_VEL
LIN {X 0,Y 698.449,Z 948.94,A -85,B 0,C 180,E1 3196.818,E2 3196.818} C_VEL
LIN {X 0,Y 698.615,Z 948.94,A -85,B 0,C 180,E1 3204.864,E2 3204.864} C_VEL
LIN {X 0,Y 698.647,Z 950.166,A -85,B 0,C 180,E1 3208.734,E2 3208.734} C_VEL
LIN {X 0,Y 705.749,Z 974.562,A -85,B 0,C 180,E1 3209.5,E2 3209.5} C_VEL
LIN {X 0,Y 704.515,Z 1041.286,A -85,B 0,C 180,E1 3211.63,E2 3211.63} C_VEL
LIN {X 0,Y 702.631,Z 1101.8,A -85,B 0,C 180,E1 3214.93,E2 3214.93} C_VEL
LIN {X 0,Y 701.043,Z 1153.302,A -85,B 0,C 180,E1 3219.248,E2 3219.248} C_VEL
LIN {X 0,Y 700.037,Z 1192.664,A -85,B 0,C 180,E1 3224.288,E2 3224.288} C_VEL
LIN {X 0,Y 699.524,Z 1218.104,A -85,B 0,C 180,E1 3229.701,E2 3229.701} C_VEL
LIN {X 0,Y 699.507,Z 1228.533,A -85,B 0,C 180,E1 3234.409,E2 3234.409} C_VEL
LIN {X 0,Y 699.603,Z 1228.636,A -85,B 0,C 180,E1 3239.391,E2 3239.391} C_VEL
LIN {X 0,Y 699.665,Z 1214.189,A -85,B 0,C 180,E1 3245.302,E2 3245.302} C_VEL
LIN {X 0,Y 699.911,Z 1185.111,A -85,B 0,C 180,E1 3250.792,E2 3250.792} C_VEL
LIN {X 0,Y 701.139,Z 1142.731,A -85,B 0,C 180,E1 3255.712,E2 3255.712} C_VEL
LIN {X 0,Y 703.039,Z 1088.9,A -85,B 0,C 180,E1 3259.82,E2 3259.82} C_VEL
LIN {X 0,Y 704.944,Z 1026.739,A -85,B 0,C 180,E1 3262.857,E2 3262.857} C_VEL
LIN {X 0,Y 703.95,Z 962.726,A -85,B 0,C 180,E1 3264.726,E2 3264.726} C_VEL
LIN {X 0,Y 699.095,Z 948.94,A -85,B 0,C 180,E1 3265.213,E2 3265.213} C_VEL
LIN {X 0,Y 698.064,Z 948.94,A -85,B 0,C 180,E1 3273.139,E2 3273.139} C_VEL
LIN {X 0,Y 697.969,Z 948.94,A -85,B 0,C 180,E1 3279.92,E2 3279.92} C_VEL
LIN {X 0,Y 698.476,Z 948.94,A -85,B 0,C 180,E1 3286.781,E2 3286.781} C_VEL
LIN {X 0,Y 698.415,Z 948.94,A -85,B 0,C 180,E1 3294.814,E2 3294.814} C_VEL
LIN {X 0,Y 698.57,Z 948.94,A -85,B 0,C 180,E1 3302.127,E2 3302.127} C_VEL
LIN {X 0,Y 698.611,Z 948.94,A -85,B 0,C 180,E1 3310.295,E2 3310.295} C_VEL
LIN {X 0,Y 699.401,Z 950.849,A -85,B 0,C 180,E1 3313.765,E2 3313.765} C_VEL
LIN {X 0,Y 701.555,Z 1024.938,A -85,B 0,C 180,E1 3314.845,E2 3314.845} C_VEL
LIN {X 0,Y 700.885,Z 1071.781,A -85,B 0,C 180,E1 3316.751,E2 3316.751} C_VEL
LIN {X 0,Y 700.103,Z 1109.974,A -85,B 0,C 180,E1 3319.669,E2 3319.669} C_VEL
LIN {X 0,Y 699.64,Z 1136.854,A -85,B 0,C 180,E1 3323.432,E2 3323.432} C_VEL
LIN {X 0,Y 699.693,Z 1148.148,A -85,B 0,C 180,E1 3326.862,E2 3326.862} C_VEL
LIN {X 0,Y 699.659,Z 1147.833,A -85,B 0,C 180,E1 3331.212,E2 3331.212} C_VEL
LIN {X 0,Y 699.675,Z 1132.718,A -85,B 0,C 180,E1 3335.257,E2 3335.257} C_VEL
LIN {X 0,Y 700.161,Z 1103.657,A -85,B 0,C 180,E1 3338.851,E2 3338.851} C_VEL
LIN {X 0,Y 700.991,Z 1063.653,A -85,B 0,C 180,E1 3341.597,E2 3341.597} C_VEL
LIN {X 0,Y 701.676,Z 1015.378,A -85,B 0,C 180,E1 3343.294,E2 3343.294} C_VEL
LIN {X 0,Y 699.1,Z 948.94,A -85,B 0,C 180,E1 3344.181,E2 3344.181} C_VEL
LIN {X 0,Y 698.315,Z 948.94,A -85,B 0,C 180,E1 3352.315,E2 3352.315} C_VEL
LIN {X 0,Y 698.735,Z 948.94,A -85,B 0,C 180,E1 3359.212,E2 3359.212} C_VEL
LIN {X 0,Y 698.391,Z 948.94,A -85,B 0,C 180,E1 3368.216,E2 3368.216} C_VEL
LIN {X 0,Y 698.528,Z 948.94,A -85,B 0,C 180,E1 3376.791,E2 3376.791} C_VEL
LIN {X 0,Y 698.411,Z 948.94,A -85,B 0,C 180,E1 3384.822,E2 3384.822} C_VEL
LIN {X 0,Y 698.548,Z 948.94,A -85,B 0,C 180,E1 3392.137,E2 3392.137} C_VEL
LIN {X 0,Y 698.811,Z 948.94,A -85,B 0,C 180,E1 3398.986,E2 3398.986} C_VEL
LIN {X 0,Y 699.449,Z 948.94,A -85,B 0,C 180,E1 3408.091,E2 3408.091} C_VEL
LIN {X 0,Y 699.173,Z 948.94,A -85,B 0,C 180,E1 3418.122,E2 3418.122} C_VEL
LIN {X 0,Y 699.139,Z 948.94,A -85,B 0,C 180,E1 3425.594,E2 3425.594} C_VEL
LIN {X 0,Y 699.047,Z 948.94,A -85,B 0,C 180,E1 3433.166,E2 3433.166} C_VEL
LIN {X 0,Y 698.545,Z 948.94,A -85,B 0,C 180,E1 3438.431,E2 3438.431} C_VEL
LIN {X 0,Y 690.694,Z 948.94,A -85,B 0,C 180,E1 3441.293,E2 3441.293} C_VEL
LIN {X 0,Y 690.792,Z 948.94,A -85,B 0,C 180,E1 3449.883,E2 3449.883} C_VEL
LIN {X 0,Y 690.613,Z 948.94,A -85,B 0,C 180,E1 3457.169,E2 3457.169} C_VEL
LIN {X 0,Y 690.339,Z 948.94,A -85,B 0,C 180,E1 3464.458,E2 3464.458} C_VEL
LIN {X 0,Y 690.728,Z 948.94,A -85,B 0,C 180,E1 3472.877,E2 3472.877} C_VEL
LIN {X 0,Y 690.817,Z 950.444,A -85,B 0,C 180,E1 3479.292,E2 3479.292} C_VEL
LIN {X 0,Y 694.11,Z 958.066,A -85,B 0,C 180,E1 3480.825,E2 3480.825} C_VEL
LIN {X 0,Y 699.585,Z 976.214,A -85,B 0,C 180,E1 3481.283,E2 3481.283} C_VEL
LIN {X 0,Y 698.811,Z 1056.579,A -85,B 0,C 180,E1 3482.543,E2 3482.543} C_VEL
LIN {X 0,Y 696.876,Z 1121.676,A -85,B 0,C 180,E1 3484.856,E2 3484.856} C_VEL
LIN {X 0,Y 694.501,Z 1181.882,A -85,B 0,C 180,E1 3488.433,E2 3488.433} C_VEL
LIN {X 0,Y 692.55,Z 1231.797,A -85,B 0,C 180,E1 3492.993,E2 3492.993} C_VEL
LIN {X 0,Y 691.408,Z 1267.552,A -85,B 0,C 180,E1 3497.999,E2 3497.999} C_VEL
LIN {X 0,Y 691.089,Z 1287.494,A -85,B 0,C 180,E1 3502.462,E2 3502.462} C_VEL
LIN {X 0,Y 691.259,Z 1298.307,A -85,B 0,C 180,E1 3507.231,E2 3507.231} C_VEL
LIN {X 0,Y 691.174,Z 1298.491,A -85,B 0,C 180,E1 3512.618,E2 3512.618} C_VEL
LIN {X 0,Y 691.16,Z 1284.952,A -85,B 0,C 180,E1 3518.235,E2 3518.235} C_VEL
LIN {X 0,Y 691.704,Z 1258.406,A -85,B 0,C 180,E1 3523.509,E2 3523.509} C_VEL
LIN {X 0,Y 693.09,Z 1217.294,A -85,B 0,C 180,E1 3528.54,E2 3528.54} C_VEL
LIN {X 0,Y 695.209,Z 1164.466,A -85,B 0,C 180,E1 3532.772,E2 3532.772} C_VEL
LIN {X 0,Y 697.495,Z 1102.437,A -85,B 0,C 180,E1 3535.972,E2 3535.972} C_VEL
LIN {X 0,Y 699.254,Z 1037.217,A -85,B 0,C 180,E1 3537.89,E2 3537.89} C_VEL
LIN {X 0,Y 697.692,Z 965.003,A -85,B 0,C 180,E1 3538.931,E2 3538.931} C_VEL
LIN {X 0,Y 693.569,Z 954.695,A -85,B 0,C 180,E1 3539.316,E2 3539.316} C_VEL
LIN {X 0,Y 690.663,Z 948.94,A -85,B 0,C 180,E1 3541.118,E2 3541.118} C_VEL
LIN {X 0,Y 690.533,Z 948.94,A -85,B 0,C 180,E1 3548.811,E2 3548.811} C_VEL
LIN {X 0,Y 690.537,Z 948.94,A -85,B 0,C 180,E1 3556.199,E2 3556.199} C_VEL
LIN {X 0,Y 690.668,Z 948.94,A -85,B 0,C 180,E1 3564.398,E2 3564.398} C_VEL
LIN {X 0,Y 690.59,Z 950.352,A -85,B 0,C 180,E1 3568.378,E2 3568.378} C_VEL
LIN {X 0,Y 698.629,Z 976.179,A -85,B 0,C 180,E1 3569.234,E2 3569.234} C_VEL
LIN {X 0,Y 697.151,Z 1042.452,A -85,B 0,C 180,E1 3571.396,E2 3571.396} C_VEL
LIN {X 0,Y 695.039,Z 1102.511,A -85,B 0,C 180,E1 3574.725,E2 3574.725} C_VEL
LIN {X 0,Y 693.224,Z 1152.923,A -85,B 0,C 180,E1 3579.003,E2 3579.003} C_VEL
LIN {X 0,Y 692.157,Z 1192.438,A -85,B 0,C 180,E1 3584.104,E2 3584.104} C_VEL
LIN {X 0,Y 691.588,Z 1217.993,A -85,B 0,C 180,E1 3589.581,E2 3589.581} C_VEL
LIN {X 0,Y 691.499,Z 1228.493,A -85,B 0,C 180,E1 3594.344,E2 3594.344} C_VEL
LIN {X 0,Y 691.592,Z 1228.668,A -85,B 0,C 180,E1 3599.384,E2 3599.384} C_VEL
LIN {X 0,Y 691.675,Z 1214.321,A -85,B 0,C 180,E1 3605.364,E2 3605.364} C_VEL
LIN {X 0,Y 691.948,Z 1185.363,A -85,B 0,C 180,E1 3610.918,E2 3610.918} C_VEL
LIN {X 0,Y 693.349,Z 1143.134,A -85,B 0,C 180,E1 3615.894,E2 3615.894} C_VEL
LIN {X 0,Y 695.492,Z 1089.474,A -85,B 0,C 180,E1 3620.044,E2 3620.044} C_VEL
LIN {X 0,Y 697.637,Z 1027.678,A -85,B 0,C 180,E1 3623.111,E2 3623.111} C_VEL
LIN {X 0,Y 696.744,Z 964.697,A -85,B 0,C 180,E1 3625,E2 3625} C_VEL
LIN {X 0,Y 691.065,Z 948.94,A -85,B 0,C 180,E1 3625.655,E2 3625.655} C_VEL
LIN {X 0,Y 690.289,Z 948.94,A -85,B 0,C 180,E1 3634.432,E2 3634.432} C_VEL
LIN {X 0,Y 690.206,Z 948.94,A -85,B 0,C 180,E1 3642.526,E2 3642.526} C_VEL
LIN {X 0,Y 690.235,Z 948.94,A -85,B 0,C 180,E1 3649.533,E2 3649.533} C_VEL
LIN {X 0,Y 690.249,Z 948.94,A -85,B 0,C 180,E1 3655.87,E2 3655.87} C_VEL
LIN {X 0,Y 690.347,Z 948.94,A -85,B 0,C 180,E1 3663.186,E2 3663.186} C_VEL
LIN {X 0,Y 690.639,Z 948.94,A -85,B 0,C 180,E1 3670.058,E2 3670.058} C_VEL
LIN {X 0,Y 691.245,Z 950.501,A -85,B 0,C 180,E1 3673.577,E2 3673.577} C_VEL
LIN {X 0,Y 693.767,Z 1024.519,A -85,B 0,C 180,E1 3674.673,E2 3674.673} C_VEL
LIN {X 0,Y 693.037,Z 1071.57,A -85,B 0,C 180,E1 3676.598,E2 3676.598} C_VEL
LIN {X 0,Y 692.196,Z 1109.85,A -85,B 0,C 180,E1 3679.55,E2 3679.55} C_VEL
LIN {X 0,Y 691.688,Z 1136.795,A -85,B 0,C 180,E1 3683.356,E2 3683.356} C_VEL
LIN {X 0,Y 691.689,Z 1148.126,A -85,B 0,C 180,E1 3686.825,E2 3686.825} C_VEL
LIN {X 0,Y 691.659,Z 1147.856,A -85,B 0,C 180,E1 3691.226,E2 3691.226} C_VEL
LIN {X 0,Y 691.682,Z 1132.786,A -85,B 0,C 180,E1 3695.318,E2 3695.318} C_VEL
LIN {X 0,Y 692.242,Z 1104.61,A -85,B 0,C 180,E1 3698.877,E2 3698.877} C_VEL
LIN {X 0,Y 693.134,Z 1063.892,A -85,B 0,C 180,E1 3701.731,E2 3701.731} C_VEL
LIN {X 0,Y 693.925,Z 1016.06,A -85,B 0,C 180,E1 3703.442,E2 3703.442} C_VEL
LIN {X 0,Y 691.661,Z 952.119,A -85,B 0,C 180,E1 3704.306,E2 3704.306} C_VEL
LIN {X 0,Y 690.927,Z 948.94,A -85,B 0,C 180,E1 3704.596,E2 3704.596} C_VEL
LIN {X 0,Y 690.223,Z 948.94,A -85,B 0,C 180,E1 3712.591,E2 3712.591} C_VEL
LIN {X 0,Y 690.519,Z 948.94,A -85,B 0,C 180,E1 3719.721,E2 3719.721} C_VEL
LIN {X 0,Y 690.606,Z 948.94,A -85,B 0,C 180,E1 3727.131,E2 3727.131} C_VEL
LIN {X 0,Y 690.613,Z 948.94,A -85,B 0,C 180,E1 3736.171,E2 3736.171} C_VEL
LIN {X 0,Y 690.514,Z 948.94,A -85,B 0,C 180,E1 3744.359,E2 3744.359} C_VEL
LIN {X 0,Y 690.617,Z 948.94,A -85,B 0,C 180,E1 3751.788,E2 3751.788} C_VEL
LIN {X 0,Y 690.493,Z 948.94,A -85,B 0,C 180,E1 3760.067,E2 3760.067} C_VEL
LIN {X 0,Y 691.422,Z 948.94,A -85,B 0,C 180,E1 3767.95,E2 3767.95} C_VEL
LIN {X 0,Y 691.177,Z 948.94,A -85,B 0,C 180,E1 3778.1,E2 3778.1} C_VEL
LIN {X 0,Y 691.107,Z 948.94,A -85,B 0,C 180,E1 3785.659,E2 3785.659} C_VEL
LIN {X 0,Y 690.979,Z 948.94,A -85,B 0,C 180,E1 3793.322,E2 3793.322} C_VEL
LIN {X 0,Y 690.694,Z 948.94,A -85,B 0,C 180,E1 3801.293,E2 3801.293} C_VEL
LIN {X 0,Y 681.977,Z 948.94,A -85,B 0,C 180,E1 3804.166,E2 3804.166} C_VEL
LIN {X 0,Y 682.659,Z 948.94,A -85,B 0,C 180,E1 3811.485,E2 3811.485} C_VEL
LIN {X 0,Y 682.485,Z 948.94,A -85,B 0,C 180,E1 3819.317,E2 3819.317} C_VEL
LIN {X 0,Y 682.114,Z 948.94,A -85,B 0,C 180,E1 3826.299,E2 3826.299} C_VEL
LIN {X 0,Y 682.766,Z 948.94,A -85,B 0,C 180,E1 3834.212,E2 3834.212} C_VEL
LIN {X 0,Y 683.001,Z 950.927,A -85,B 0,C 180,E1 3838.635,E2 3838.635} C_VEL
LIN {X 0,Y 689.734,Z 966.414,A -85,B 0,C 180,E1 3840.719,E2 3840.719} C_VEL
LIN {X 0,Y 692.562,Z 985.65,A -85,B 0,C 180,E1 3841.074,E2 3841.074} C_VEL
LIN {X 0,Y 691.565,Z 1060.322,A -85,B 0,C 180,E1 3842.334,E2 3842.334} C_VEL
LIN {X 0,Y 689.407,Z 1124.509,A -85,B 0,C 180,E1 3844.707,E2 3844.707} C_VEL
LIN {X 0,Y 686.781,Z 1184.196,A -85,B 0,C 180,E1 3848.362,E2 3848.362} C_VEL
LIN {X 0,Y 684.661,Z 1233.198,A -85,B 0,C 180,E1 3852.957,E2 3852.957} C_VEL
LIN {X 0,Y 683.489,Z 1267.556,A -85,B 0,C 180,E1 3857.858,E2 3857.858} C_VEL
LIN {X 0,Y 683.151,Z 1287.495,A -85,B 0,C 180,E1 3862.374,E2 3862.374} C_VEL
LIN {X 0,Y 683.445,Z 1297.844,A -85,B 0,C 180,E1 3866.85,E2 3866.85} C_VEL
LIN {X 0,Y 683.511,Z 1299.147,A -85,B 0,C 180,E1 3871.94,E2 3871.94} C_VEL
LIN {X 0,Y 683.394,Z 1287.254,A -85,B 0,C 180,E1 3877.687,E2 3877.687} C_VEL
LIN {X 0,Y 683.823,Z 1260.622,A -85,B 0,C 180,E1 3883.318,E2 3883.318} C_VEL
LIN {X 0,Y 685.27,Z 1220.3,A -85,B 0,C 180,E1 3888.448,E2 3888.448} C_VEL
LIN {X 0,Y 687.505,Z 1168.725,A -85,B 0,C 180,E1 3892.753,E2 3892.753} C_VEL
LIN {X 0,Y 690.051,Z 1107.385,A -85,B 0,C 180,E1 3896.067,E2 3896.067} C_VEL
LIN {X 0,Y 692.049,Z 1041.224,A -85,B 0,C 180,E1 3898.122,E2 3898.122} C_VEL
LIN {X 0,Y 690.844,Z 967.774,A -85,B 0,C 180,E1 3899.213,E2 3899.213} C_VEL
LIN {X 0,Y 689.077,Z 961.096,A -85,B 0,C 180,E1 3899.733,E2 3899.733} C_VEL
LIN {X 0,Y 682.504,Z 948.94,A -85,B 0,C 180,E1 3901.79,E2 3901.79} C_VEL
LIN {X 0,Y 682.252,Z 948.94,A -85,B 0,C 180,E1 3909.888,E2 3909.888} C_VEL
LIN {X 0,Y 682.282,Z 948.94,A -85,B 0,C 180,E1 3917.29,E2 3917.29} C_VEL
LIN {X 0,Y 682.474,Z 948.94,A -85,B 0,C 180,E1 3925.466,E2 3925.466} C_VEL
LIN {X 0,Y 682.521,Z 950.451,A -85,B 0,C 180,E1 3928.01,E2 3928.01} C_VEL
LIN {X 0,Y 691.5,Z 977.71,A -85,B 0,C 180,E1 3928.963,E2 3928.963} C_VEL
LIN {X 0,Y 689.791,Z 1043.497,A -85,B 0,C 180,E1 3931.152,E2 3931.152} C_VEL
LIN {X 0,Y 687.442,Z 1103.177,A -85,B 0,C 180,E1 3934.512,E2 3934.512} C_VEL
LIN {X 0,Y 685.383,Z 1154.169,A -85,B 0,C 180,E1 3938.922,E2 3938.922} C_VEL
LIN {X 0,Y 684.245,Z 1192.211,A -85,B 0,C 180,E1 3943.915,E2 3943.915} C_VEL
LIN {X 0,Y 683.658,Z 1217.881,A -85,B 0,C 180,E1 3949.459,E2 3949.459} C_VEL
LIN {X 0,Y 683.469,Z 1228.454,A -85,B 0,C 180,E1 3954.277,E2 3954.277} C_VEL
LIN {X 0,Y 683.582,Z 1228.701,A -85,B 0,C 180,E1 3959.376,E2 3959.376} C_VEL
LIN {X 0,Y 683.79,Z 1215.612,A -85,B 0,C 180,E1 3965.106,E2 3965.106} C_VEL
LIN {X 0,Y 684.088,Z 1187.78,A -85,B 0,C 180,E1 3970.722,E2 3970.722} C_VEL
LIN {X 0,Y 685.5,Z 1146.942,A -85,B 0,C 180,E1 3975.735,E2 3975.735} C_VEL
LIN {X 0,Y 687.788,Z 1093.97,A -85,B 0,C 180,E1 3980.015,E2 3980.015} C_VEL
LIN {X 0,Y 690.161,Z 1032.787,A -85,B 0,C 180,E1 3983.204,E2 3983.204} C_VEL
LIN {X 0,Y 690.034,Z 968.11,A -85,B 0,C 180,E1 3985.231,E2 3985.231} C_VEL
LIN {X 0,Y 683.058,Z 948.94,A -85,B 0,C 180,E1 3985.932,E2 3985.932} C_VEL
LIN {X 0,Y 682.313,Z 948.94,A -85,B 0,C 180,E1 3994.574,E2 3994.574} C_VEL
LIN {X 0,Y 682.233,Z 948.94,A -85,B 0,C 180,E1 4002.748,E2 4002.748} C_VEL
LIN {X 0,Y 682.403,Z 948.94,A -85,B 0,C 180,E1 4010.638,E2 4010.638} C_VEL
LIN {X 0,Y 682.604,Z 948.94,A -85,B 0,C 180,E1 4018.902,E2 4018.902} C_VEL
LIN {X 0,Y 682.911,Z 948.94,A -85,B 0,C 180,E1 4028.461,E2 4028.461} C_VEL
LIN {X 0,Y 683.066,Z 949.938,A -85,B 0,C 180,E1 4033.383,E2 4033.383} C_VEL
LIN {X 0,Y 686.056,Z 1022.273,A -85,B 0,C 180,E1 4034.45,E2 4034.45} C_VEL
LIN {X 0,Y 685.25,Z 1069.972,A -85,B 0,C 180,E1 4036.361,E2 4036.361} C_VEL
LIN {X 0,Y 684.38,Z 1108.149,A -85,B 0,C 180,E1 4039.268,E2 4039.268} C_VEL
LIN {X 0,Y 683.853,Z 1135.158,A -85,B 0,C 180,E1 4042.959,E2 4042.959} C_VEL
LIN {X 0,Y 683.679,Z 1148.103,A -85,B 0,C 180,E1 4046.788,E2 4046.788} C_VEL
LIN {X 0,Y 683.663,Z 1147.957,A -85,B 0,C 180,E1 4051.199,E2 4051.199} C_VEL
LIN {X 0,Y 683.686,Z 1132.855,A -85,B 0,C 180,E1 4055.381,E2 4055.381} C_VEL
LIN {X 0,Y 684.29,Z 1104.686,A -85,B 0,C 180,E1 4058.986,E2 4058.986} C_VEL
LIN {X 0,Y 685.301,Z 1064.13,A -85,B 0,C 180,E1 4061.867,E2 4061.867} C_VEL
LIN {X 0,Y 686.171,Z 1016.803,A -85,B 0,C 180,E1 4063.592,E2 4063.592} C_VEL
LIN {X 0,Y 683.81,Z 953.027,A -85,B 0,C 180,E1 4064.477,E2 4064.477} C_VEL
LIN {X 0,Y 682.879,Z 948.94,A -85,B 0,C 180,E1 4064.744,E2 4064.744} C_VEL
LIN {X 0,Y 682.241,Z 948.94,A -85,B 0,C 180,E1 4072.559,E2 4072.559} C_VEL
LIN {X 0,Y 682.422,Z 948.94,A -85,B 0,C 180,E1 4079.981,E2 4079.981} C_VEL
LIN {X 0,Y 682.388,Z 948.94,A -85,B 0,C 180,E1 4087.831,E2 4087.831} C_VEL
LIN {X 0,Y 682.6,Z 948.94,A -85,B 0,C 180,E1 4096.208,E2 4096.208} C_VEL
LIN {X 0,Y 682.546,Z 948.94,A -85,B 0,C 180,E1 4104.177,E2 4104.177} C_VEL
LIN {X 0,Y 682.615,Z 948.94,A -85,B 0,C 180,E1 4111.427,E2 4111.427} C_VEL
LIN {X 0,Y 682.538,Z 948.94,A -85,B 0,C 180,E1 4119.824,E2 4119.824} C_VEL
LIN {X 0,Y 683.427,Z 948.94,A -85,B 0,C 180,E1 4127.807,E2 4127.807} C_VEL
LIN {X 0,Y 683.183,Z 948.94,A -85,B 0,C 180,E1 4138.078,E2 4138.078} C_VEL
LIN {X 0,Y 683.058,Z 948.94,A -85,B 0,C 180,E1 4145.726,E2 4145.726} C_VEL
LIN {X 0,Y 682.882,Z 948.94,A -85,B 0,C 180,E1 4153.483,E2 4153.483} C_VEL
LIN {X 0,Y 682.588,Z 948.94,A -85,B 0,C 180,E1 4161.511,E2 4161.511} C_VEL
LIN {X 0,Y 681.977,Z 948.94,A -85,B 0,C 180,E1 4164.166,E2 4164.166} C_VEL
LIN {X 0,Y 674.477,Z 948.94,A -85,B 0,C 180,E1 4167.103,E2 4167.103} C_VEL
LIN {X 0,Y 674.902,Z 948.94,A -85,B 0,C 180,E1 4174.978,E2 4174.978} C_VEL
LIN {X 0,Y 674.623,Z 948.94,A -85,B 0,C 180,E1 4183.313,E2 4183.313} C_VEL
LIN {X 0,Y 674.739,Z 948.94,A -85,B 0,C 180,E1 4191.842,E2 4191.842} C_VEL
LIN {X 0,Y 675.013,Z 950.601,A -85,B 0,C 180,E1 4198.267,E2 4198.267} C_VEL
LIN {X 0,Y 685.137,Z 974.173,A -85,B 0,C 180,E1 4200.595,E2 4200.595} C_VEL
LIN {X 0,Y 684.552,Z 1056.414,A -85,B 0,C 180,E1 4201.916,E2 4201.916} C_VEL
LIN {X 0,Y 682.154,Z 1121.75,A -85,B 0,C 180,E1 4204.278,E2 4204.278} C_VEL
LIN {X 0,Y 679.37,Z 1180.969,A -85,B 0,C 180,E1 4207.857,E2 4207.857} C_VEL
LIN {X 0,Y 677.083,Z 1230.335,A -85,B 0,C 180,E1 4212.424,E2 4212.424} C_VEL
LIN {X 0,Y 675.667,Z 1265.692,A -85,B 0,C 180,E1 4217.386,E2 4217.386} C_VEL
LIN {X 0,Y 675.199,Z 1287.495,A -85,B 0,C 180,E1 4222.283,E2 4222.283} C_VEL
LIN {X 0,Y 675.478,Z 1297.847,A -85,B 0,C 180,E1 4226.813,E2 4226.813} C_VEL
LIN {X 0,Y 675.507,Z 1299.149,A -85,B 0,C 180,E1 4231.963,E2 4231.963} C_VEL
LIN {X 0,Y 675.363,Z 1287.253,A -85,B 0,C 180,E1 4237.779,E2 4237.779} C_VEL
LIN {X 0,Y 675.9,Z 1261.422,A -85,B 0,C 180,E1 4243.343,E2 4243.343} C_VEL
LIN {X 0,Y 677.429,Z 1222.005,A -85,B 0,C 180,E1 4248.488,E2 4248.488} C_VEL
LIN {X 0,Y 679.938,Z 1169.756,A -85,B 0,C 180,E1 4252.949,E2 4252.949} C_VEL
LIN {X 0,Y 682.773,Z 1108.134,A -85,B 0,C 180,E1 4256.334,E2 4256.334} C_VEL
LIN {X 0,Y 684.968,Z 1042.307,A -85,B 0,C 180,E1 4258.414,E2 4258.414} C_VEL
LIN {X 0,Y 684.062,Z 970.049,A -85,B 0,C 180,E1 4259.542,E2 4259.542} C_VEL
LIN {X 0,Y 675.094,Z 951.884,A -85,B 0,C 180,E1 4261.602,E2 4261.602} C_VEL
LIN {X 0,Y 674.471,Z 948.94,A -85,B 0,C 180,E1 4261.952,E2 4261.952} C_VEL
LIN {X 0,Y 674.245,Z 948.94,A -85,B 0,C 180,E1 4269.933,E2 4269.933} C_VEL
LIN {X 0,Y 674.33,Z 948.94,A -85,B 0,C 180,E1 4277.039,E2 4277.039} C_VEL
LIN {X 0,Y 674.505,Z 948.94,A -85,B 0,C 180,E1 4285.246,E2 4285.246} C_VEL
LIN {X 0,Y 674.492,Z 950.501,A -85,B 0,C 180,E1 4287.634,E2 4287.634} C_VEL
LIN {X 0,Y 684.382,Z 979.713,A -85,B 0,C 180,E1 4288.697,E2 4288.697} C_VEL
LIN {X 0,Y 682.349,Z 1046.753,A -85,B 0,C 180,E1 4291.005,E2 4291.005} C_VEL
LIN {X 0,Y 679.713,Z 1106.412,A -85,B 0,C 180,E1 4294.482,E2 4294.482} C_VEL
LIN {X 0,Y 677.542,Z 1155.815,A -85,B 0,C 180,E1 4298.88,E2 4298.88} C_VEL
LIN {X 0,Y 676.215,Z 1193.955,A -85,B 0,C 180,E1 4304.054,E2 4304.054} C_VEL
LIN {X 0,Y 675.589,Z 1218.742,A -85,B 0,C 180,E1 4309.659,E2 4309.659} C_VEL
LIN {X 0,Y 675.13,Z 1229.545,A -85,B 0,C 180,E1 4315.5,E2 4315.5} C_VEL
LIN {X 0,Y 675.225,Z 1227.118,A -85,B 0,C 180,E1 4320.657,E2 4320.657} C_VEL
LIN {X 0,Y 675.448,Z 1212.143,A -85,B 0,C 180,E1 4326.14,E2 4326.14} C_VEL
LIN {X 0,Y 676.019,Z 1183.675,A -85,B 0,C 180,E1 4331.507,E2 4331.507} C_VEL
LIN {X 0,Y 677.844,Z 1142.206,A -85,B 0,C 180,E1 4336.434,E2 4336.434} C_VEL
LIN {X 0,Y 680.511,Z 1088.769,A -85,B 0,C 180,E1 4340.629,E2 4340.629} C_VEL
LIN {X 0,Y 683.218,Z 1026.429,A -85,B 0,C 180,E1 4343.758,E2 4343.758} C_VEL
LIN {X 0,Y 682.605,Z 969.596,A -85,B 0,C 180,E1 4345.537,E2 4345.537} C_VEL
LIN {X 0,Y 675.043,Z 948.94,A -85,B 0,C 180,E1 4346.343,E2 4346.343} C_VEL
LIN {X 0,Y 674.393,Z 948.94,A -85,B 0,C 180,E1 4355.039,E2 4355.039} C_VEL
LIN {X 0,Y 674.376,Z 948.94,A -85,B 0,C 180,E1 4363.368,E2 4363.368} C_VEL
LIN {X 0,Y 674.527,Z 948.94,A -85,B 0,C 180,E1 4371.747,E2 4371.747} C_VEL
LIN {X 0,Y 674.613,Z 948.94,A -85,B 0,C 180,E1 4381.046,E2 4381.046} C_VEL
LIN {X 0,Y 674.694,Z 948.94,A -85,B 0,C 180,E1 4389.566,E2 4389.566} C_VEL
LIN {X 0,Y 675.053,Z 950.533,A -85,B 0,C 180,E1 4393.197,E2 4393.197} C_VEL
LIN {X 0,Y 678.529,Z 1008.442,A -85,B 0,C 180,E1 4393.973,E2 4393.973} C_VEL
LIN {X 0,Y 677.651,Z 1057.176,A -85,B 0,C 180,E1 4395.544,E2 4395.544} C_VEL
LIN {X 0,Y 676.515,Z 1099.466,A -85,B 0,C 180,E1 4398.323,E2 4398.323} C_VEL
LIN {X 0,Y 675.7,Z 1129.639,A -85,B 0,C 180,E1 4401.9,E2 4401.9} C_VEL
LIN {X 0,Y 675.553,Z 1146.805,A -85,B 0,C 180,E1 4406.105,E2 4406.105} C_VEL
LIN {X 0,Y 675.788,Z 1148.894,A -85,B 0,C 180,E1 4410.611,E2 4410.611} C_VEL
LIN {X 0,Y 675.887,Z 1136.27,A -85,B 0,C 180,E1 4414.797,E2 4414.797} C_VEL
LIN {X 0,Y 676.419,Z 1110.28,A -85,B 0,C 180,E1 4418.536,E2 4418.536} C_VEL
LIN {X 0,Y 677.38,Z 1071.648,A -85,B 0,C 180,E1 4421.598,E2 4421.598} C_VEL
LIN {X 0,Y 678.253,Z 1025.204,A -85,B 0,C 180,E1 4423.552,E2 4423.552} C_VEL
LIN {X 0,Y 676.235,Z 954.698,A -85,B 0,C 180,E1 4424.638,E2 4424.638} C_VEL
LIN {X 0,Y 674.889,Z 948.94,A -85,B 0,C 180,E1 4424.781,E2 4424.781} C_VEL
LIN {X 0,Y 674.485,Z 948.94,A -85,B 0,C 180,E1 4431.754,E2 4431.754} C_VEL
LIN {X 0,Y 674.305,Z 948.94,A -85,B 0,C 180,E1 4440.379,E2 4440.379} C_VEL
LIN {X 0,Y 674.284,Z 948.94,A -85,B 0,C 180,E1 4448.188,E2 4448.188} C_VEL
LIN {X 0,Y 674.453,Z 948.94,A -85,B 0,C 180,E1 4456.934,E2 4456.934} C_VEL
LIN {X 0,Y 674.33,Z 948.94,A -85,B 0,C 180,E1 4465.156,E2 4465.156} C_VEL
LIN {X 0,Y 674.417,Z 948.94,A -85,B 0,C 180,E1 4472.635,E2 4472.635} C_VEL
LIN {X 0,Y 674.562,Z 948.94,A -85,B 0,C 180,E1 4479.575,E2 4479.575} C_VEL
LIN {X 0,Y 675.421,Z 948.94,A -85,B 0,C 180,E1 4487.661,E2 4487.661} C_VEL
LIN {X 0,Y 675.198,Z 948.94,A -85,B 0,C 180,E1 4498.055,E2 4498.055} C_VEL
LIN {X 0,Y 675.037,Z 948.94,A -85,B 0,C 180,E1 4505.795,E2 4505.795} C_VEL
LIN {X 0,Y 674.79,Z 948.94,A -85,B 0,C 180,E1 4513.648,E2 4513.648} C_VEL
LIN {X 0,Y 674.489,Z 948.94,A -85,B 0,C 180,E1 4521.782,E2 4521.782} C_VEL
LIN {X 0,Y 674.477,Z 948.94,A -85,B 0,C 180,E1 4527.103,E2 4527.103} C_VEL
LIN {X 0,Y 666.664,Z 948.94,A -85,B 0,C 180,E1 4530.076,E2 4530.076} C_VEL
LIN {X 0,Y 666.508,Z 948.94,A -85,B 0,C 180,E1 4538.297,E2 4538.297} C_VEL
LIN {X 0,Y 666.103,Z 948.94,A -85,B 0,C 180,E1 4546.039,E2 4546.039} C_VEL
LIN {X 0,Y 666.683,Z 948.94,A -85,B 0,C 180,E1 4553.9,E2 4553.9} C_VEL
LIN {X 0,Y 667.049,Z 950.341,A -85,B 0,C 180,E1 4557.923,E2 4557.923} C_VEL
LIN {X 0,Y 678.602,Z 977.497,A -85,B 0,C 180,E1 4560.323,E2 4560.323} C_VEL
LIN {X 0,Y 677.442,Z 1057.585,A -85,B 0,C 180,E1 4561.627,E2 4561.627} C_VEL
LIN {X 0,Y 674.816,Z 1122.77,A -85,B 0,C 180,E1 4564.031,E2 4564.031} C_VEL
LIN {X 0,Y 671.709,Z 1182.594,A -85,B 0,C 180,E1 4567.723,E2 4567.723} C_VEL
LIN {X 0,Y 669.193,Z 1231.799,A -85,B 0,C 180,E1 4572.381,E2 4572.381} C_VEL
LIN {X 0,Y 667.639,Z 1267.564,A -85,B 0,C 180,E1 4577.565,E2 4577.565} C_VEL
LIN {X 0,Y 666.981,Z 1289.44,A -85,B 0,C 180,E1 4582.845,E2 4582.845} C_VEL
LIN {X 0,Y 666.948,Z 1299.204,A -85,B 0,C 180,E1 4588.077,E2 4588.077} C_VEL
LIN {X 0,Y 666.927,Z 1297.766,A -85,B 0,C 180,E1 4593.293,E2 4593.293} C_VEL
LIN {X 0,Y 667.146,Z 1284.945,A -85,B 0,C 180,E1 4598.534,E2 4598.534} C_VEL
LIN {X 0,Y 667.869,Z 1259.471,A -85,B 0,C 180,E1 4603.833,E2 4603.833} C_VEL
LIN {X 0,Y 669.671,Z 1220.532,A -85,B 0,C 180,E1 4608.87,E2 4608.87} C_VEL
LIN {X 0,Y 672.463,Z 1168.737,A -85,B 0,C 180,E1 4613.291,E2 4613.291} C_VEL
LIN {X 0,Y 675.528,Z 1108.135,A -85,B 0,C 180,E1 4616.638,E2 4616.638} C_VEL
LIN {X 0,Y 677.959,Z 1041.551,A -85,B 0,C 180,E1 4618.753,E2 4618.753} C_VEL
LIN {X 0,Y 678.027,Z 974.377,A -85,B 0,C 180,E1 4619.798,E2 4619.798} C_VEL
LIN {X 0,Y 667.306,Z 953.634,A -85,B 0,C 180,E1 4621.579,E2 4621.579} C_VEL
LIN {X 0,Y 666.5,Z 948.94,A -85,B 0,C 180,E1 4621.923,E2 4621.923} C_VEL
LIN {X 0,Y 666.172,Z 948.94,A -85,B 0,C 180,E1 4630.517,E2 4630.517} C_VEL
LIN {X 0,Y 666.145,Z 948.94,A -85,B 0,C 180,E1 4637.8,E2 4637.8} C_VEL
LIN {X 0,Y 666.338,Z 948.94,A -85,B 0,C 180,E1 4646.271,E2 4646.271} C_VEL
LIN {X 0,Y 666.576,Z 950.953,A -85,B 0,C 180,E1 4647.272,E2 4647.272} C_VEL
LIN {X 0,Y 677.304,Z 983.268,A -85,B 0,C 180,E1 4648.467,E2 4648.467} C_VEL
LIN {X 0,Y 674.914,Z 1049.886,A -85,B 0,C 180,E1 4650.854,E2 4650.854} C_VEL
LIN {X 0,Y 672.018,Z 1108.723,A -85,B 0,C 180,E1 4654.389,E2 4654.389} C_VEL
LIN {X 0,Y 669.684,Z 1158.714,A -85,B 0,C 180,E1 4658.992,E2 4658.992} C_VEL
LIN {X 0,Y 668.161,Z 1195.698,A -85,B 0,C 180,E1 4664.195,E2 4664.195} C_VEL
LIN {X 0,Y 667.659,Z 1218.631,A -85,B 0,C 180,E1 4669.535,E2 4669.535} C_VEL
LIN {X 0,Y 667.137,Z 1229.519,A -85,B 0,C 180,E1 4675.446,E2 4675.446} C_VEL
LIN {X 0,Y 667.219,Z 1227.176,A -85,B 0,C 180,E1 4680.664,E2 4680.664} C_VEL
LIN {X 0,Y 667.463,Z 1212.276,A -85,B 0,C 180,E1 4686.214,E2 4686.214} C_VEL
LIN {X 0,Y 668.102,Z 1184.115,A -85,B 0,C 180,E1 4691.617,E2 4691.617} C_VEL
LIN {X 0,Y 670.073,Z 1142.61,A -85,B 0,C 180,E1 4696.63,E2 4696.63} C_VEL
LIN {X 0,Y 673.02,Z 1088.539,A -85,B 0,C 180,E1 4700.924,E2 4700.924} C_VEL
LIN {X 0,Y 675.997,Z 1026.328,A -85,B 0,C 180,E1 4704.072,E2 4704.072} C_VEL
LIN {X 0,Y 675.533,Z 971.812,A -85,B 0,C 180,E1 4705.816,E2 4705.816} C_VEL
LIN {X 0,Y 667.044,Z 948.94,A -85,B 0,C 180,E1 4706.743,E2 4706.743} C_VEL
LIN {X 0,Y 666.389,Z 948.94,A -85,B 0,C 180,E1 4716.017,E2 4716.017} C_VEL
LIN {X 0,Y 666.483,Z 948.94,A -85,B 0,C 180,E1 4725.855,E2 4725.855} C_VEL
LIN {X 0,Y 666.394,Z 948.94,A -85,B 0,C 180,E1 4734.468,E2 4734.468} C_VEL
LIN {X 0,Y 666.454,Z 948.94,A -85,B 0,C 180,E1 4742.143,E2 4742.143} C_VEL
LIN {X 0,Y 666.722,Z 948.94,A -85,B 0,C 180,E1 4749.311,E2 4749.311} C_VEL
LIN {X 0,Y 667.066,Z 950.862,A -85,B 0,C 180,E1 4752.997,E2 4752.997} C_VEL
LIN {X 0,Y 670.817,Z 992.077,A -85,B 0,C 180,E1 4753.544,E2 4753.544} C_VEL
LIN {X 0,Y 670.161,Z 1042.708,A -85,B 0,C 180,E1 4754.748,E2 4754.748} C_VEL
LIN {X 0,Y 668.837,Z 1087.871,A -85,B 0,C 180,E1 4757.242,E2 4757.242} C_VEL
LIN {X 0,Y 667.668,Z 1121.854,A -85,B 0,C 180,E1 4760.649,E2 4760.649} C_VEL
LIN {X 0,Y 667.258,Z 1142.042,A -85,B 0,C 180,E1 4764.422,E2 4764.422} C_VEL
LIN {X 0,Y 667.167,Z 1149.63,A -85,B 0,C 180,E1 4768.013,E2 4768.013} C_VEL
LIN {X 0,Y 667.331,Z 1146.607,A -85,B 0,C 180,E1 4771.922,E2 4771.922} C_VEL
LIN {X 0,Y 667.609,Z 1131.146,A -85,B 0,C 180,E1 4775.838,E2 4775.838} C_VEL
LIN {X 0,Y 668.397,Z 1101.743,A -85,B 0,C 180,E1 4779.509,E2 4779.509} C_VEL
LIN {X 0,Y 669.657,Z 1059.953,A -85,B 0,C 180,E1 4782.397,E2 4782.397} C_VEL
LIN {X 0,Y 670.86,Z 1011.694,A -85,B 0,C 180,E1 4784.061,E2 4784.061} C_VEL
LIN {X 0,Y 668.504,Z 955.93,A -85,B 0,C 180,E1 4784.82,E2 4784.82} C_VEL
LIN {X 0,Y 666.796,Z 948.94,A -85,B 0,C 180,E1 4784.991,E2 4784.991} C_VEL
LIN {X 0,Y 666.168,Z 948.94,A -85,B 0,C 180,E1 4792.634,E2 4792.634} C_VEL
LIN {X 0,Y 666.179,Z 948.94,A -85,B 0,C 180,E1 4800.79,E2 4800.79} C_VEL
LIN {X 0,Y 666.181,Z 948.94,A -85,B 0,C 180,E1 4808.738,E2 4808.738} C_VEL
LIN {X 0,Y 666.518,Z 948.94,A -85,B 0,C 180,E1 4815.991,E2 4815.991} C_VEL
LIN {X 0,Y 666.354,Z 948.94,A -85,B 0,C 180,E1 4824.475,E2 4824.475} C_VEL
LIN {X 0,Y 666.43,Z 948.94,A -85,B 0,C 180,E1 4832.153,E2 4832.153} C_VEL
LIN {X 0,Y 666.626,Z 948.94,A -85,B 0,C 180,E1 4839.321,E2 4839.321} C_VEL
LIN {X 0,Y 667.412,Z 948.94,A -85,B 0,C 180,E1 4847.51,E2 4847.51} C_VEL
LIN {X 0,Y 667.201,Z 948.94,A -85,B 0,C 180,E1 4858.032,E2 4858.032} C_VEL
LIN {X 0,Y 666.99,Z 948.94,A -85,B 0,C 180,E1 4865.865,E2 4865.865} C_VEL
LIN {X 0,Y 666.707,Z 948.94,A -85,B 0,C 180,E1 4873.817,E2 4873.817} C_VEL
LIN {X 0,Y 666.374,Z 948.94,A -85,B 0,C 180,E1 4882.061,E2 4882.061} C_VEL
LIN {X 0,Y 666.664,Z 948.94,A -85,B 0,C 180,E1 4890.076,E2 4890.076} C_VEL
LIN {X 0,Y 658.656,Z 948.94,A -85,B 0,C 180,E1 4893.055,E2 4893.055} C_VEL
LIN {X 0,Y 658.581,Z 948.94,A -85,B 0,C 180,E1 4901.567,E2 4901.567} C_VEL
LIN {X 0,Y 658.654,Z 948.94,A -85,B 0,C 180,E1 4910.734,E2 4910.734} C_VEL
LIN {X 0,Y 659.09,Z 950.598,A -85,B 0,C 180,E1 4917.607,E2 4917.607} C_VEL
LIN {X 0,Y 670.014,Z 976.283,A -85,B 0,C 180,E1 4919.878,E2 4919.878} C_VEL
LIN {X 0,Y 670.338,Z 1058.759,A -85,B 0,C 180,E1 4921.333,E2 4921.333} C_VEL
LIN {X 0,Y 667.414,Z 1124.726,A -85,B 0,C 180,E1 4923.824,E2 4923.824} C_VEL
LIN {X 0,Y 664.083,Z 1183.586,A -85,B 0,C 180,E1 4927.535,E2 4927.535} C_VEL
LIN {X 0,Y 661.328,Z 1233.102,A -85,B 0,C 180,E1 4932.327,E2 4932.327} C_VEL
LIN {X 0,Y 659.633,Z 1269.171,A -85,B 0,C 180,E1 4937.72,E2 4937.72} C_VEL
LIN {X 0,Y 659.022,Z 1289.438,A -85,B 0,C 180,E1 4942.758,E2 4942.758} C_VEL
LIN {X 0,Y 658.971,Z 1299.206,A -85,B 0,C 180,E1 4948.053,E2 4948.053} C_VEL
LIN {X 0,Y 658.944,Z 1297.769,A -85,B 0,C 180,E1 4953.333,E2 4953.333} C_VEL
LIN {X 0,Y 659.136,Z 1284.942,A -85,B 0,C 180,E1 4958.638,E2 4958.638} C_VEL
LIN {X 0,Y 659.942,Z 1259.467,A -85,B 0,C 180,E1 4964.003,E2 4964.003} C_VEL
LIN {X 0,Y 661.911,Z 1220.536,A -85,B 0,C 180,E1 4969.1,E2 4969.1} C_VEL
LIN {X 0,Y 664.938,Z 1168.743,A -85,B 0,C 180,E1 4973.571,E2 4973.571} C_VEL
LIN {X 0,Y 668.325,Z 1107.088,A -85,B 0,C 180,E1 4976.994,E2 4976.994} C_VEL
LIN {X 0,Y 670.946,Z 1041.621,A -85,B 0,C 180,E1 4979.081,E2 4979.081} C_VEL
LIN {X 0,Y 670.244,Z 976.072,A -85,B 0,C 180,E1 4980.128,E2 4980.128} C_VEL
LIN {X 0,Y 658.654,Z 950.67,A -85,B 0,C 180,E1 4981.727,E2 4981.727} C_VEL
LIN {X 0,Y 658.267,Z 948.94,A -85,B 0,C 180,E1 4989.448,E2 4989.448} C_VEL
LIN {X 0,Y 658.185,Z 948.94,A -85,B 0,C 180,E1 4997.152,E2 4997.152} C_VEL
LIN {X 0,Y 658.344,Z 948.94,A -85,B 0,C 180,E1 5005.624,E2 5005.624} C_VEL
LIN {X 0,Y 658.494,Z 950.697,A -85,B 0,C 180,E1 5007,E2 5007} C_VEL
LIN {X 0,Y 670.234,Z 985.51,A -85,B 0,C 180,E1 5008.197,E2 5008.197} C_VEL
LIN {X 0,Y 667.563,Z 1051.105,A -85,B 0,C 180,E1 5010.606,E2 5010.606} C_VEL
LIN {X 0,Y 664.368,Z 1110.672,A -85,B 0,C 180,E1 5014.27,E2 5014.27} C_VEL
LIN {X 0,Y 661.798,Z 1160.255,A -85,B 0,C 180,E1 5018.954,E2 5018.954} C_VEL
LIN {X 0,Y 660.103,Z 1197.362,A -85,B 0,C 180,E1 5024.339,E2 5024.339} C_VEL
LIN {X 0,Y 659.331,Z 1220.459,A -85,B 0,C 180,E1 5030.071,E2 5030.071} C_VEL
LIN {X 0,Y 659.159,Z 1229.493,A -85,B 0,C 180,E1 5035.39,E2 5035.39} C_VEL
LIN {X 0,Y 659.224,Z 1227.233,A -85,B 0,C 180,E1 5040.673,E2 5040.673} C_VEL
LIN {X 0,Y 659.469,Z 1212.409,A -85,B 0,C 180,E1 5046.289,E2 5046.289} C_VEL
LIN {X 0,Y 660.203,Z 1184.256,A -85,B 0,C 180,E1 5051.774,E2 5051.774} C_VEL
LIN {X 0,Y 662.322,Z 1143.012,A -85,B 0,C 180,E1 5056.831,E2 5056.831} C_VEL
LIN {X 0,Y 665.537,Z 1089.38,A -85,B 0,C 180,E1 5061.152,E2 5061.152} C_VEL
LIN {X 0,Y 668.744,Z 1027.488,A -85,B 0,C 180,E1 5064.34,E2 5064.34} C_VEL
LIN {X 0,Y 668.654,Z 974.798,A -85,B 0,C 180,E1 5066.065,E2 5066.065} C_VEL
LIN {X 0,Y 659.02,Z 948.94,A -85,B 0,C 180,E1 5067.072,E2 5067.072} C_VEL
LIN {X 0,Y 658.38,Z 948.94,A -85,B 0,C 180,E1 5077.285,E2 5077.285} C_VEL
LIN {X 0,Y 658.323,Z 948.94,A -85,B 0,C 180,E1 5086.592,E2 5086.592} C_VEL
LIN {X 0,Y 658.319,Z 948.94,A -85,B 0,C 180,E1 5094.955,E2 5094.955} C_VEL
LIN {X 0,Y 658.304,Z 948.94,A -85,B 0,C 180,E1 5103.256,E2 5103.256} C_VEL
LIN {X 0,Y 658.544,Z 948.94,A -85,B 0,C 180,E1 5110.449,E2 5110.449} C_VEL
LIN {X 0,Y 658.92,Z 950.563,A -85,B 0,C 180,E1 5112.782,E2 5112.782} C_VEL
LIN {X 0,Y 663.129,Z 987.848,A -85,B 0,C 180,E1 5113.304,E2 5113.304} C_VEL
LIN {X 0,Y 662.659,Z 1038.053,A -85,B 0,C 180,E1 5114.377,E2 5114.377} C_VEL
LIN {X 0,Y 661.3,Z 1083.191,A -85,B 0,C 180,E1 5116.703,E2 5116.703} C_VEL
LIN {X 0,Y 659.954,Z 1118.113,A -85,B 0,C 180,E1 5120.038,E2 5120.038} C_VEL
LIN {X 0,Y 659.34,Z 1140.791,A -85,B 0,C 180,E1 5124.023,E2 5124.023} C_VEL
LIN {X 0,Y 659.177,Z 1149.62,A -85,B 0,C 180,E1 5127.989,E2 5127.989} C_VEL
LIN {X 0,Y 659.331,Z 1146.636,A -85,B 0,C 180,E1 5131.946,E2 5131.946} C_VEL
LIN {X 0,Y 659.62,Z 1131.218,A -85,B 0,C 180,E1 5135.909,E2 5135.909} C_VEL
LIN {X 0,Y 660.575,Z 1100.765,A -85,B 0,C 180,E1 5139.776,E2 5139.776} C_VEL
LIN {X 0,Y 661.949,Z 1059.204,A -85,B 0,C 180,E1 5142.644,E2 5142.644} C_VEL
LIN {X 0,Y 663.219,Z 1010.55,A -85,B 0,C 180,E1 5144.278,E2 5144.278} C_VEL
LIN {X 0,Y 660.639,Z 956.468,A -85,B 0,C 180,E1 5145.017,E2 5145.017} C_VEL
LIN {X 0,Y 658.694,Z 948.94,A -85,B 0,C 180,E1 5145.327,E2 5145.327} C_VEL
LIN {X 0,Y 658.288,Z 948.94,A -85,B 0,C 180,E1 5152.317,E2 5152.317} C_VEL
LIN {X 0,Y 658.308,Z 948.94,A -85,B 0,C 180,E1 5160.137,E2 5160.137} C_VEL
LIN {X 0,Y 658.357,Z 948.94,A -85,B 0,C 180,E1 5167.601,E2 5167.601} C_VEL
LIN {X 0,Y 658.414,Z 948.94,A -85,B 0,C 180,E1 5176.496,E2 5176.496} C_VEL
LIN {X 0,Y 658.301,Z 948.94,A -85,B 0,C 180,E1 5184.85,E2 5184.85} C_VEL
LIN {X 0,Y 658.386,Z 948.94,A -85,B 0,C 180,E1 5192.458,E2 5192.458} C_VEL
LIN {X 0,Y 658.397,Z 948.94,A -85,B 0,C 180,E1 5200.458,E2 5200.458} C_VEL
LIN {X 0,Y 659.394,Z 948.94,A -85,B 0,C 180,E1 5208.704,E2 5208.704} C_VEL
LIN {X 0,Y 659.22,Z 948.94,A -85,B 0,C 180,E1 5218.008,E2 5218.008} C_VEL
LIN {X 0,Y 658.944,Z 948.94,A -85,B 0,C 180,E1 5225.937,E2 5225.937} C_VEL
LIN {X 0,Y 658.646,Z 948.94,A -85,B 0,C 180,E1 5233.989,E2 5233.989} C_VEL
LIN {X 0,Y 658.31,Z 948.94,A -85,B 0,C 180,E1 5242.346,E2 5242.346} C_VEL
LIN {X 0,Y 658.644,Z 948.94,A -85,B 0,C 180,E1 5251.216,E2 5251.216} C_VEL
LIN {X 0,Y 658.656,Z 948.94,A -85,B 0,C 180,E1 5253.055,E2 5253.055} C_VEL
LIN {X 0,Y 650.598,Z 948.94,A -85,B 0,C 180,E1 5256.09,E2 5256.09} C_VEL
LIN {X 0,Y 650.245,Z 948.94,A -85,B 0,C 180,E1 5264.675,E2 5264.675} C_VEL
LIN {X 0,Y 650.644,Z 948.94,A -85,B 0,C 180,E1 5273.569,E2 5273.569} C_VEL
LIN {X 0,Y 650.981,Z 950.175,A -85,B 0,C 180,E1 5277.225,E2 5277.225} C_VEL
LIN {X 0,Y 661.162,Z 977.934,A -85,B 0,C 180,E1 5279.459,E2 5279.459} C_VEL
LIN {X 0,Y 664.719,Z 987.132,A -85,B 0,C 180,E1 5279.754,E2 5279.754} C_VEL
LIN {X 0,Y 663.161,Z 1061.811,A -85,B 0,C 180,E1 5281.088,E2 5281.088} C_VEL
LIN {X 0,Y 660.039,Z 1126.682,A -85,B 0,C 180,E1 5283.613,E2 5283.613} C_VEL
LIN {X 0,Y 656.415,Z 1185.085,A -85,B 0,C 180,E1 5287.383,E2 5287.383} C_VEL
LIN {X 0,Y 653.474,Z 1234.144,A -85,B 0,C 180,E1 5292.24,E2 5292.24} C_VEL
LIN {X 0,Y 651.723,Z 1268.813,A -85,B 0,C 180,E1 5297.498,E2 5297.498} C_VEL
LIN {X 0,Y 651.055,Z 1289.436,A -85,B 0,C 180,E1 5302.669,E2 5302.669} C_VEL
LIN {X 0,Y 650.976,Z 1299.209,A -85,B 0,C 180,E1 5308.029,E2 5308.029} C_VEL
LIN {X 0,Y 650.938,Z 1297.773,A -85,B 0,C 180,E1 5313.374,E2 5313.374} C_VEL
LIN {X 0,Y 651.158,Z 1284.94,A -85,B 0,C 180,E1 5318.745,E2 5318.745} C_VEL
LIN {X 0,Y 652.036,Z 1259.462,A -85,B 0,C 180,E1 5324.176,E2 5324.176} C_VEL
LIN {X 0,Y 654.173,Z 1220.537,A -85,B 0,C 180,E1 5329.334,E2 5329.334} C_VEL
LIN {X 0,Y 657.425,Z 1168.749,A -85,B 0,C 180,E1 5333.857,E2 5333.857} C_VEL
LIN {X 0,Y 661.167,Z 1107.088,A -85,B 0,C 180,E1 5337.311,E2 5337.311} C_VEL
LIN {X 0,Y 663.812,Z 1042.645,A -85,B 0,C 180,E1 5339.377,E2 5339.377} C_VEL
LIN {X 0,Y 662.382,Z 979.106,A -85,B 0,C 180,E1 5340.306,E2 5340.306} C_VEL
LIN {X 0,Y 650.692,Z 951.225,A -85,B 0,C 180,E1 5341.683,E2 5341.683} C_VEL
LIN {X 0,Y 650.397,Z 948.94,A -85,B 0,C 180,E1 5342.408,E2 5342.408} C_VEL
LIN {X 0,Y 650.108,Z 948.94,A -85,B 0,C 180,E1 5350.664,E2 5350.664} C_VEL
LIN {X 0,Y 650.011,Z 948.94,A -85,B 0,C 180,E1 5358.298,E2 5358.298} C_VEL
LIN {X 0,Y 650.341,Z 948.946,A -85,B 0,C 180,E1 5366.703,E2 5366.703} C_VEL
LIN {X 0,Y 663.08,Z 988.657,A -85,B 0,C 180,E1 5367.948,E2 5367.948} C_VEL
LIN {X 0,Y 660.202,Z 1053.12,A -85,B 0,C 180,E1 5370.392,E2 5370.392} C_VEL
LIN {X 0,Y 656.74,Z 1112.219,A -85,B 0,C 180,E1 5374.117,E2 5374.117} C_VEL
LIN {X 0,Y 653.906,Z 1161.861,A -85,B 0,C 180,E1 5378.928,E2 5378.928} C_VEL
LIN {X 0,Y 652.064,Z 1198.935,A -85,B 0,C 180,E1 5384.487,E2 5384.487} C_VEL
LIN {X 0,Y 651.386,Z 1220.349,A -85,B 0,C 180,E1 5389.949,E2 5389.949} C_VEL
LIN {X 0,Y 651.163,Z 1229.466,A -85,B 0,C 180,E1 5395.334,E2 5395.334} C_VEL
LIN {X 0,Y 651.218,Z 1227.29,A -85,B 0,C 180,E1 5400.681,E2 5400.681} C_VEL
LIN {X 0,Y 651.462,Z 1212.542,A -85,B 0,C 180,E1 5406.367,E2 5406.367} C_VEL
LIN {X 0,Y 652.29,Z 1185.022,A -85,B 0,C 180,E1 5411.841,E2 5411.841} C_VEL
LIN {X 0,Y 654.592,Z 1143.461,A -85,B 0,C 180,E1 5417.031,E2 5417.031} C_VEL
LIN {X 0,Y 658.054,Z 1089.946,A -85,B 0,C 180,E1 5421.404,E2 5421.404} C_VEL
LIN {X 0,Y 661.543,Z 1028.297,A -85,B 0,C 180,E1 5424.628,E2 5424.628} C_VEL
LIN {X 0,Y 661.429,Z 976.885,A -85,B 0,C 180,E1 5426.344,E2 5426.344} C_VEL
LIN {X 0,Y 650.973,Z 948.94,A -85,B 0,C 180,E1 5427.459,E2 5427.459} C_VEL
LIN {X 0,Y 650.389,Z 948.94,A -85,B 0,C 180,E1 5436.535,E2 5436.535} C_VEL
LIN {X 0,Y 650.4,Z 948.94,A -85,B 0,C 180,E1 5445.397,E2 5445.397} C_VEL
LIN {X 0,Y 650.474,Z 948.94,A -85,B 0,C 180,E1 5453.634,E2 5453.634} C_VEL
LIN {X 0,Y 650.456,Z 948.94,A -85,B 0,C 180,E1 5461.395,E2 5461.395} C_VEL
LIN {X 0,Y 650.57,Z 948.94,A -85,B 0,C 180,E1 5470.2,E2 5470.2} C_VEL
LIN {X 0,Y 650.864,Z 950.488,A -85,B 0,C 180,E1 5472.565,E2 5472.565} C_VEL
LIN {X 0,Y 655.36,Z 983.975,A -85,B 0,C 180,E1 5473.061,E2 5473.061} C_VEL
LIN {X 0,Y 655.015,Z 1036.897,A -85,B 0,C 180,E1 5474.126,E2 5474.126} C_VEL
LIN {X 0,Y 653.678,Z 1081.505,A -85,B 0,C 180,E1 5476.374,E2 5476.374} C_VEL
LIN {X 0,Y 652.236,Z 1117.679,A -85,B 0,C 180,E1 5479.75,E2 5479.75} C_VEL
LIN {X 0,Y 651.396,Z 1141.295,A -85,B 0,C 180,E1 5483.95,E2 5483.95} C_VEL
LIN {X 0,Y 651.188,Z 1149.915,A -85,B 0,C 180,E1 5487.964,E2 5487.964} C_VEL
LIN {X 0,Y 651.34,Z 1147.044,A -85,B 0,C 180,E1 5491.969,E2 5491.969} C_VEL
LIN {X 0,Y 651.724,Z 1130.217,A -85,B 0,C 180,E1 5496.316,E2 5496.316} C_VEL
LIN {X 0,Y 652.778,Z 1100.635,A -85,B 0,C 180,E1 5500.006,E2 5500.006} C_VEL
LIN {X 0,Y 654.245,Z 1060.378,A -85,B 0,C 180,E1 5502.795,E2 5502.795} C_VEL
LIN {X 0,Y 655.535,Z 1012.034,A -85,B 0,C 180,E1 5504.45,E2 5504.45} C_VEL
LIN {X 0,Y 653.315,Z 958.997,A -85,B 0,C 180,E1 5505.183,E2 5505.183} C_VEL
LIN {X 0,Y 650.65,Z 948.94,A -85,B 0,C 180,E1 5505.521,E2 5505.521} C_VEL
LIN {X 0,Y 650.151,Z 948.94,A -85,B 0,C 180,E1 5512.725,E2 5512.725} C_VEL
LIN {X 0,Y 650.319,Z 948.94,A -85,B 0,C 180,E1 5520.069,E2 5520.069} C_VEL
LIN {X 0,Y 650.133,Z 948.94,A -85,B 0,C 180,E1 5528.526,E2 5528.526} C_VEL
LIN {X 0,Y 650.293,Z 948.94,A -85,B 0,C 180,E1 5537.255,E2 5537.255} C_VEL
LIN {X 0,Y 650.261,Z 948.94,A -85,B 0,C 180,E1 5545.104,E2 5545.104} C_VEL
LIN {X 0,Y 650.317,Z 948.94,A -85,B 0,C 180,E1 5552.913,E2 5552.913} C_VEL
LIN {X 0,Y 650.371,Z 948.94,A -85,B 0,C 180,E1 5560.779,E2 5560.779} C_VEL
LIN {X 0,Y 651.386,Z 948.94,A -85,B 0,C 180,E1 5568.563,E2 5568.563} C_VEL
LIN {X 0,Y 651.222,Z 948.94,A -85,B 0,C 180,E1 5577.983,E2 5577.983} C_VEL
LIN {X 0,Y 650.901,Z 948.94,A -85,B 0,C 180,E1 5586.01,E2 5586.01} C_VEL
LIN {X 0,Y 650.407,Z 948.94,A -85,B 0,C 180,E1 5594.64,E2 5594.64} C_VEL
LIN {X 0,Y 650.212,Z 948.94,A -85,B 0,C 180,E1 5602.64,E2 5602.64} C_VEL
LIN {X 0,Y 650.704,Z 948.94,A -85,B 0,C 180,E1 5610.084,E2 5610.084} C_VEL
LIN {X 0,Y 650.598,Z 948.94,A -85,B 0,C 180,E1 5616.09,E2 5616.09} C_VEL
LIN {X 0,Y 642.427,Z 948.94,A -85,B 0,C 180,E1 5619.155,E2 5619.155} C_VEL
LIN {X 0,Y 642.279,Z 948.94,A -85,B 0,C 180,E1 5628.087,E2 5628.087} C_VEL
LIN {X 0,Y 642.826,Z 949.06,A -85,B 0,C 180,E1 5636.778,E2 5636.778} C_VEL
LIN {X 0,Y 651.212,Z 976.495,A -85,B 0,C 180,E1 5638.918,E2 5638.918} C_VEL
LIN {X 0,Y 657.81,Z 989.597,A -85,B 0,C 180,E1 5639.43,E2 5639.43} C_VEL
LIN {X 0,Y 655.971,Z 1062.298,A -85,B 0,C 180,E1 5640.787,E2 5640.787} C_VEL
LIN {X 0,Y 652.721,Z 1127.368,A -85,B 0,C 180,E1 5643.331,E2 5643.331} C_VEL
LIN {X 0,Y 648.842,Z 1185.72,A -85,B 0,C 180,E1 5647.158,E2 5647.158} C_VEL
LIN {X 0,Y 645.757,Z 1233.35,A -85,B 0,C 180,E1 5651.92,E2 5651.92} C_VEL
LIN {X 0,Y 643.789,Z 1269.003,A -85,B 0,C 180,E1 5657.378,E2 5657.378} C_VEL
LIN {X 0,Y 643.09,Z 1289.434,A -85,B 0,C 180,E1 5662.578,E2 5662.578} C_VEL
LIN {X 0,Y 643.009,Z 1299.211,A -85,B 0,C 180,E1 5668.005,E2 5668.005} C_VEL
LIN {X 0,Y 642.954,Z 1297.776,A -85,B 0,C 180,E1 5673.416,E2 5673.416} C_VEL
LIN {X 0,Y 643.153,Z 1284.937,A -85,B 0,C 180,E1 5678.854,E2 5678.854} C_VEL
LIN {X 0,Y 644.137,Z 1259.457,A -85,B 0,C 180,E1 5684.354,E2 5684.354} C_VEL
